// Device/Application/CAN_Rx/CAN0_RX_Inverters
(* VERSION V1_0  *)

FUNCTION_BLOCK CAN0_RX_Inverters
VAR_INPUT
END_VAR
VAR_OUTPUT	
(*INVERTER 1*)
	(* AMK_Actual_Values_1_INV1, ID=283*)
		AMK_bSystemReady1_CAN: BOOL;
		AMK_bError1_CAN: BOOL;
		AMK_bWarn1_CAN: BOOL;
		AMK_bQuitDcOn1_CAN: BOOL;
		AMK_bDcOn1_check_CAN: BOOL;
		AMK_bQuitInverterOn1_CAN: BOOL;
		AMK_bInverterOn1_check_CAN: BOOL;
		AMK_bDerating1_CAN: BOOL;
		AMK_ActualVelocity1_CAN: INT;
		AMK_TorqueCurrent1_CAN: INT;
		AMK_MagnetizingCurrent1_CAN: INT;
	(* AMK_Actual_Values_2_INV1, ID=285*)
		AMK_TempMotor1_CAN: INT;
		AMK_TempInverter1_CAN: INT;
		AMK_ErrorInfo1_CAN: UINT;
		AMK_TempIGBT1_CAN: INT;
(*INVERTER 2*)
	(* AMK_Actual_Values_1_INV2, ID=284*)
		AMK_bSystemReady2_CAN: BOOL;
		AMK_bError2_CAN: BOOL;
		AMK_bWarn2_CAN: BOOL;
		AMK_bQuitDcOn2_CAN: BOOL;
		AMK_bDcOn2_check_CAN: BOOL;
		AMK_bQuitInverterOn2_CAN: BOOL;
		AMK_bInverterOn2_check_CAN: BOOL;
		AMK_bDerating2_CAN: BOOL;
		AMK_ActualVelocity2_CAN: INT;
		AMK_TorqueCurrent2_CAN: INT;
		AMK_MagnetizingCurrent2_CAN: INT;
	(* AMK_Actual_Values_2_INV2, ID=286*)	
		AMK_TempMotor2_CAN: INT;
		AMK_TempInverter2_CAN: INT;
		AMK_ErrorInfo2_CAN: UINT;
		AMK_TempIGBT2_CAN: INT;
(*INVERTER 3*)
	(* AMK_Actual_Values_1_INV3, ID=287*)
		AMK_bSystemReady3_CAN: BOOL;
		AMK_bError3_CAN: BOOL;
		AMK_bWarn3_CAN: BOOL;
		AMK_bQuitDcOn3_CAN: BOOL;
		AMK_bDcOn3_check_CAN: BOOL;
		AMK_bQuitInverterOn3_CAN: BOOL;
		AMK_bInverterOn3_check_CAN: BOOL;
		AMK_bDerating3_CAN: BOOL;
		AMK_ActualVelocity3_CAN: INT;
		AMK_TorqueCurrent3_CAN: INT;
		AMK_MagnetizingCurrent3_CAN: INT;
	(* AMK_Actual_Values_2_INV3, ID=289*)
		AMK_TempMotor3_CAN: INT;
		AMK_TempInverter3_CAN: INT;
		AMK_ErrorInfo3_CAN: UINT;
		AMK_TempIGBT3_CAN: INT;
(*INVERTER 4*)
	(* AMK_Actual_Values_1_INV4, ID=288*)
		AMK_bSystemReady4_CAN: BOOL;
		AMK_bError4_CAN: BOOL;
		AMK_bWarn4_CAN: BOOL;
		AMK_bQuitDcOn4_CAN: BOOL;
		AMK_bDcOn4_check_CAN: BOOL;
		AMK_bQuitInverterOn4_CAN: BOOL;
		AMK_bInverterOn4_check_CAN: BOOL;
		AMK_bDerating4_CAN: BOOL;
		AMK_ActualVelocity4_CAN: INT;
		AMK_TorqueCurrent4_CAN: INT;
		AMK_MagnetizingCurrent4_CAN: INT;
	(* AMK_Actual_Values_2_INV4, ID=290*)
		AMK_TempMotor4_CAN: INT;
		AMK_TempInverter4_CAN: INT;
		AMK_ErrorInfo4_CAN: UINT;
		AMK_TempIGBT4_CAN: INT;
		
		(*
(*DATA_LOGGER*)
		DL_Msg_Cntr_CAN: SINT;
		DL_Status_CAN: SINT;
		DL_Power_CAN: INT;
		DL_Voltage_CAN: INT;
		DL_Current_CAN: INT;
		
(*BATTERY*)
	BatCurrent_MSB_CAN: INT;
	BatVoltage_MSB_CAN: INT;
	BatSoc_CAN: INT;
	BatSoh_CAN: INT;
	BatState_CAN: INT;
	BatAlmLv_CAN: INT;
	BatLife_CAN: INT;
	MaxCellVolt_MSB_CAN: INT;
	MinCellVolt_MSB_CAN: INT;
	MaxCellVoltNO_CAN: INT;
	MinCellVoltNO_CAN: INT;
	MaxTemp_CAN: INT;
	MinTemp_CAN: INT;
	MaxTempNo_CAN: INT;
	MinTempNo_CAN: INT;
	CoolingCtl_CAN: INT;
	HeatingCtl_CAN: INT;
	PosRlyStr_CAN: INT;
	NegRlyStr_CAN: INT;
	PreRlyStr_CAN: INT;
	OnChrRlyStr_CAN: INT;
	OffChrRlyStr_CAN: INT;
	ChrState_CAN: INT;
	ChrCommunication_CAN: BOOL;
	ChrOFFCC2_CAN: BOOL;
	ChrONCC_CAN: INT;
	ChrReqVolt_MSB_CAN: INT;
	ChrReqCurr_MSB_CAN: INT;
	MaxChrCurtLimit_MSB_CAN: INT;
	MaxDisCurtLimit_MSB_CAN: INT;
	MaxChrPowerLimit_MSB_CAN: INT;
	MaxDisPowerLimit_MSB_CAN: INT;
	ALM_CELL_OV_CAN: INT;
	ALM_CELL_UV_CAN: INT;
	ALM_CELL_OT_CAN: INT;
	ALM_CELL_UT_CAN: INT;
	ALM_CELL_LBK_CAN: BOOL;
	ALM_CELL_TBK_CAN: BOOL;
	ALM_BATT_DV_CAN: INT;
	ALM_BATT_DT_CAN: INT;
	ALM_BATT_OV_CAN: INT;
	ALM_BATT_UV_CAN: INT;
	ALM_BATT_OC_CAN: INT;
	ALM_BATT_UC_CAN: INT;
	ALM_CHRG_OCS_CAN: INT;
	ALM_DSCH_OCS_CAN: INT;
	ALM_CHRG_OCT_CAN: INT;
	ALM_DSCH_OCT_CAN: INT;
	ALM_BSU_OFFLINE_CAN: INT;
	ALM_BSU_FAULT_CAN: BOOL;
	ALM_LEAK_OC_CAN: INT;
	ALM_PRECHRG_FAIL_CAN: BOOL;
	ALM_AUX_FAIL_CAN: BOOL;
	ALM_BMU_FAIL_CAN: BOOL;
	ALM_VCU_OFFLINE_CAN: INT;
	ALM_HVREL_FAIL_CAN: BOOL;
	ALM_HALL_BREAK_CAN: BOOL;
	CellVoltN_1_CAN: INT;
	CellVoltN_2_CAN: INT;
	CellVoltN_3_CAN: INT;
	CellVoltN_4_CAN: INT;
	CellVoltN_5_CAN: INT;
	CellVoltN_6_CAN: INT;
	CellVoltN_7_CAN: INT;
	CellVoltN_8_CAN: INT;
	CellVoltN_9_CAN: INT;
	CellVoltN_10_CAN: INT;
	CellVoltN_11_CAN: INT;
	CellVoltN_12_CAN: INT;
	CellVoltN_13_CAN: INT;
	CellVoltN_14_CAN: INT;
	CellVoltN_15_CAN: INT;
	CellVoltN_16_CAN: INT;
	CellVoltN_17_CAN: INT;
	CellVoltN_18_CAN: INT;
	CellVoltN_19_CAN: INT;
	CellVoltN_20_CAN: INT;
	CellVoltN_21_CAN: INT;
	CellVoltN_22_CAN: INT;
	CellVoltN_23_CAN: INT;
	CellVoltN_24_CAN: INT;
	CellVoltN_25_CAN: INT;
	CellVoltN_26_CAN: INT;
	CellVoltN_27_CAN: INT;
	CellVoltN_28_CAN: INT;
	CellVoltN_29_CAN: INT;
	CellVoltN_30_CAN: INT;
	CellVoltN_31_CAN: INT;
	CellVoltN_32_CAN: INT;
	CellVoltN_33_CAN: INT;
	CellVoltN_34_CAN: INT;
	CellVoltN_35_CAN: INT;
	CellVoltN_36_CAN: INT;
	CellVoltN_37_CAN: INT;
	CellVoltN_38_CAN: INT;
	CellVoltN_39_CAN: INT;
	CellVoltN_40_CAN: INT;
	CellVoltN_41_CAN: INT;
	CellVoltN_42_CAN: INT;
	CellVoltN_43_CAN: INT;
	CellVoltN_44_CAN: INT;
	CellVoltN_45_CAN: INT;
	CellVoltN_46_CAN: INT;
	CellVoltN_47_CAN: INT;
	CellVoltN_48_CAN: INT;
	CellVoltN_49_CAN: INT;
	CellVoltN_50_CAN: INT;
	CellVoltN_51_CAN: INT;
	CellVoltN_52_CAN: INT;
	CellVoltN_53_CAN: INT;
	CellVoltN_54_CAN: INT;
	CellVoltN_55_CAN: INT;
	CellVoltN_56_CAN: INT;
	CellVoltN_57_CAN: INT;
	CellVoltN_58_CAN: INT;
	CellVoltN_59_CAN: INT;
	CellVoltN_60_CAN: INT;
	CellVoltN_61_CAN: INT;
	CellVoltN_62_CAN: INT;
	CellVoltN_63_CAN: INT;
	CellVoltN_64_CAN: INT;
	CellVoltN_65_CAN: INT;
	CellVoltN_66_CAN: INT;
	CellVoltN_67_CAN: INT;
	CellVoltN_68_CAN: INT;
	CellVoltN_69_CAN: INT;
	CellVoltN_70_CAN: INT;
	CellVoltN_71_CAN: INT;
	CellVoltN_72_CAN: INT;
	CellVoltN_73_CAN: INT;
	CellVoltN_74_CAN: INT;
	CellVoltN_75_CAN: INT;
	CellVoltN_76_CAN: INT;
	CellVoltN_77_CAN: INT;
	CellVoltN_78_CAN: INT;
	CellVoltN_79_CAN: INT;
	CellVoltN_80_CAN: INT;
	CellVoltN_81_CAN: INT;
	CellVoltN_82_CAN: INT;
	CellVoltN_83_CAN: INT;
	CellVoltN_84_CAN: INT;
	CellVoltN_85_CAN: INT;
	CellVoltN_86_CAN: INT;
	CellVoltN_87_CAN: INT;
	CellVoltN_88_CAN: INT;
	CellVoltN_89_CAN: INT;
	CellVoltN_90_CAN: INT;
	CellVoltN_91_CAN: INT;
	CellVoltN_92_CAN: INT;
	CellVoltN_93_CAN: INT;
	CellVoltN_94_CAN: INT;
	CellVoltN_95_CAN: INT;
	CellVoltN_96_CAN: INT;
	CellVoltN_97_CAN: INT;
	CellVoltN_98_CAN: INT;
	CellVoltN_99_CAN: INT;
	CellVoltN_100_CAN: INT;
	CellVoltN_101_CAN: INT;
	CellVoltN_102_CAN: INT;
	CellVoltN_103_CAN: INT;
	CellVoltN_104_CAN: INT;
	CellVoltN_105_CAN: INT;
	CellVoltN_106_CAN: INT;
	CellVoltN_107_CAN: INT;
	CellVoltN_108_CAN: INT;
	CellVoltN_109_CAN: INT;
	CellVoltN_110_CAN: INT;
	CellVoltN_111_CAN: INT;
	CellVoltN_112_CAN: INT;
	CellVoltN_113_CAN: INT;
	CellVoltN_114_CAN: INT;
	CellVoltN_115_CAN: INT;
	CellVoltN_116_CAN: INT;
	CellVoltN_117_CAN: INT;
	CellVoltN_118_CAN: INT;
	CellVoltN_119_CAN: INT;
	CellVoltN_120_CAN: INT;
	CellVoltN_121_CAN: INT;
	CellVoltN_122_CAN: INT;
	CellVoltN_123_CAN: INT;
	CellVoltN_124_CAN: INT;
	CellVoltN_125_CAN: INT;
	CellVoltN_126_CAN: INT;
	CellVoltN_127_CAN: INT;
	CellVoltN_128_CAN: INT;
	CellVoltN_129_CAN: INT;
	CellVoltN_130_CAN: INT;
	CellVoltN_131_CAN: INT;
	CellVoltN_132_CAN: INT;
	CellVoltN_133_CAN: INT;
	CellVoltN_134_CAN: INT;
	CellVoltN_135_CAN: INT;
	CellVoltN_136_CAN: INT;
	CellVoltN_137_CAN: INT;
	CellVoltN_138_CAN: INT;
	CellTempN_1_CAN: INT;
	CellTempN_2_CAN: INT;
	CellTempN_3_CAN: INT;
	CellTempN_4_CAN: INT;
	CellTempN_5_CAN: INT;
	CellTempN_6_CAN: INT;
	CellTempN_7_CAN: INT;
	CellTempN_8_CAN: INT;
	CellTempN_9_CAN: INT;
	CellTempN_10_CAN: INT;
	CellTempN_11_CAN: INT;
	CellTempN_12_CAN: INT;
	CellTempN_13_CAN: INT;
	CellTempN_14_CAN: INT;
	CellTempN_15_CAN: INT;
	CellTempN_16_CAN: INT;
	CellTempN_17_CAN: INT;
	CellTempN_18_CAN: INT;
	CellTempN_19_CAN: INT;
	CellTempN_20_CAN: INT;
	CellTempN_21_CAN: INT;
	CellTempN_22_CAN: INT;
	CellTempN_23_CAN: INT;
	CellTempN_24_CAN: INT;
	CellTempN_25_CAN: INT;
	CellTempN_26_CAN: INT;
	CellTempN_27_CAN: INT;
	CellTempN_28_CAN: INT;
	CellTempN_29_CAN: INT;
	CellTempN_30_CAN: INT;
	CellTempN_31_CAN: INT;
	CellTempN_32_CAN: INT;
	CellTempN_33_CAN: INT;
	CellTempN_34_CAN: INT;
	CellTempN_35_CAN: INT;
	CellTempN_36_CAN: INT;
	CellTempN_37_CAN: INT;
	CellTempN_38_CAN: INT;
	CellTempN_39_CAN: INT;
	CellTempN_40_CAN: INT;
	CellTempN_41_CAN: INT;
	CellTempN_42_CAN: INT;
	CellTempN_43_CAN: INT;
	CellTempN_44_CAN: INT;
	CellTempN_45_CAN: INT;
	CellTempN_46_CAN: INT;
	CellTempN_47_CAN: INT;
	CellTempN_48_CAN: INT;
	CellTempN_49_CAN: INT;
	CellTempN_50_CAN: INT;
	CellTempN_51_CAN: INT;
	CellTempN_52_CAN: INT;
	CellTempN_53_CAN: INT;
	CellTempN_54_CAN: INT;
	CellTempN_55_CAN: INT;
	CellTempN_56_CAN: INT;
	CellTempN_57_CAN: INT;
	CellTempN_58_CAN: INT;
	CellTempN_59_CAN: INT;
	CellTempN_60_CAN: INT;
	MainRlyCmd_CAN: INT;
	ShutDownCmd_CAN: INT;
	BMS_State_CAN: DINT;
	*)
			
END_VAR
VAR
(*CanRx*)
	(* INVERTER_1*)
		FBRX_AMK_Actual_Values_1_INV1: CanRx;
		FBRX_AMK_Actual_Values_2_INV1: CanRx;
	(* INVERTER_2*)
		FBRX_AMK_Actual_Values_1_INV2:CanRx;
		FBRX_AMK_Actual_Values_2_INV2:CanRx;
	(* INVERTER_3*)
		FBRX_AMK_Actual_Values_1_INV3:CanRx;
		FBRX_AMK_Actual_Values_2_INV3:CanRx;
	(* INVERTER_4*)
		FBRX_AMK_Actual_Values_1_INV4:CanRx;
		FBRX_AMK_Actual_Values_2_INV4:CanRx;
		
		(*
	(*BATTERY*)
		FBRX_BATTERY:CanRx;
	(*DATA_LOGGER*)	
		FBRX_DATA_LOGGER:CanRx;
		
		(*BATTERY*)
		FBRX_BMS_HCU_INFO:CanRx;
		FBRX_BMS_HCU_MAXV: CanRx;
		FBRX_BMS_HCU_MAXT: CanRx;
		FBRX_BMS_HCU_RELAY: CanRx;
		FBRX_BMS_HCU_POWER: CanRx;
		FBRX_BMS_HCU_ALARM: CanRx;
		FBRX_BMS_HCU_CMD: CanRx;
		FBRX_BMS_HCU_CELLV_1: CanRx;
		FBRX_BMS_HCU_CELLV_2: CanRx;
		FBRX_BMS_HCU_CELLV_3: CanRx;
		FBRX_BMS_HCU_CELLV_4: CanRx;
		FBRX_BMS_HCU_CELLV_5: CanRx;
		FBRX_BMS_HCU_CELLV_6: CanRx;
		FBRX_BMS_HCU_CELLV_7: CanRx;
		FBRX_BMS_HCU_CELLV_8: CanRx;
		FBRX_BMS_HCU_CELLV_9: CanRx;
		FBRX_BMS_HCU_CELLV_10: CanRx;
		FBRX_BMS_HCU_CELLV_11: CanRx;
		FBRX_BMS_HCU_CELLV_12: CanRx;
		FBRX_BMS_HCU_CELLV_13: CanRx;
		FBRX_BMS_HCU_CELLV_14: CanRx;
		FBRX_BMS_HCU_CELLV_15: CanRx;
		FBRX_BMS_HCU_CELLV_16: CanRx;
		FBRX_BMS_HCU_CELLV_17: CanRx;
		FBRX_BMS_HCU_CELLV_18: CanRx;
		FBRX_BMS_HCU_CELLV_19: CanRx;
		FBRX_BMS_HCU_CELLV_20: CanRx;
		FBRX_BMS_HCU_CELLV_21: CanRx;
		FBRX_BMS_HCU_CELLV_22: CanRx;
		FBRX_BMS_HCU_CELLV_23: CanRx;
		FBRX_BMS_HCU_CELLV_24: CanRx;
		FBRX_BMS_HCU_CELLV_25: CanRx;
		FBRX_BMS_HCU_CELLV_26: CanRx;
		FBRX_BMS_HCU_CELLV_27: CanRx;
		FBRX_BMS_HCU_CELLV_28: CanRx;
		FBRX_BMS_HCU_CELLV_29: CanRx;
		FBRX_BMS_HCU_CELLV_30: CanRx;
		FBRX_BMS_HCU_CELLV_31: CanRx;
		FBRX_BMS_HCU_CELLV_32: CanRx;
		FBRX_BMS_HCU_CELLV_33: CanRx;
		FBRX_BMS_HCU_CELLV_34: CanRx;
		FBRX_BMS_HCU_CELLV_35: CanRx;
		FBRX_BMS_HCU_CELLT_1: CanRx;
		FBRX_BMS_HCU_CELLT_2: CanRx;
		FBRX_BMS_HCU_CELLT_3: CanRx;
		FBRX_BMS_HCU_CELLT_4: CanRx;
		FBRX_BMS_HCU_CELLT_5: CanRx;
		FBRX_BMS_HCU_CELLT_6: CanRx;
		FBRX_BMS_HCU_CELLT_7: CanRx;
		FBRX_BMS_HCU_CELLT_8: CanRx;
		FBRX_Battery_status: CanRx;
		*)
		
(*Time_out_Counter*)
	(* INVERTER_1*)
		Counter_time_out_AMK_Actual_Values_1_INV1:INT:=0;
		Counter_time_out_AMK_Actual_Values_2_INV1:INT:=0;
	(* INVERTER_2*)	
		Counter_time_out_AMK_Actual_Values_1_INV2:INT:=0;
		Counter_time_out_AMK_Actual_Values_2_INV2:INT:=0;
	(* INVERTER_3*)	
		Counter_time_out_AMK_Actual_Values_1_INV3:INT:=0;
		Counter_time_out_AMK_Actual_Values_2_INV3:INT:=0;
	(* INVERTER_4*)	
		Counter_time_out_AMK_Actual_Values_1_INV4:INT:=0;
		Counter_time_out_AMK_Actual_Values_2_INV4:INT:=0;
		(*
	(*battery*)
		Counter_time_out_BATTERY:INT:=0;
		Counter_time_out_FBRX_BMS_HCU_INFO:INT:=0;
	(*DATA_LOGGER*)
		Counter_time_out_DATA_LOGGER:INT:=0;	
		
		*)
		
		
END_VAR

(*--------------------------------------------------INVERTER_1_RX--------------------------------------------------*)
	(* AMK_Actual_Values_1_INV1, ID=283*)
		FBRX_AMK_Actual_Values_1_INV1 (	iCAN			:= ADR(GVL.H_CAN_RX_0),  				(* Structure for sending / receiving CAN messages *)
								iCanId				:= 16#283,							(* CAN Id of receiving message *) 
								iCanIdExtended		:= FALSE,  							(* Standard CAN Frame *)
								iTimeoutLimit		:= T#500MS,							(* Timeout after 500ms - Flag will be set *) 
								oByteCount			=> , 
								oData				=> , 
								oNewData			=> , 
								oCanTimeout			=> , 
								oReceiverId			=> , 
								oTooManyReceivers	=> );	
				
								
				IF FBRX_AMK_Actual_Values_1_INV1  .oNewData THEN											(* If new CAN data is available *)
						AMK_bSystemReady1_CAN:=FBRX_AMK_Actual_Values_1_INV1.oData[1].0;
						AMK_bError1_CAN:=FBRX_AMK_Actual_Values_1_INV1.oData[1].1;
						AMK_bWarn1_CAN:=FBRX_AMK_Actual_Values_1_INV1.oData[1].2;
						AMK_bQuitDcOn1_CAN:=FBRX_AMK_Actual_Values_1_INV1.oData[1].3;
						AMK_bDcOn1_check_CAN:=FBRX_AMK_Actual_Values_1_INV1.oData[1].4;
						AMK_bQuitInverterOn1_CAN:=FBRX_AMK_Actual_Values_1_INV1.oData[1].5;
						AMK_bInverterOn1_check_CAN:=FBRX_AMK_Actual_Values_1_INV1.oData[1].6;
						AMK_bDerating1_CAN:=FBRX_AMK_Actual_Values_1_INV1.oData[1].7;
						AMK_ActualVelocity1_CAN:=FBRX_AMK_Actual_Values_1_INV1.oData[2]+SHL(BYTE_TO_INT(FBRX_AMK_Actual_Values_1_INV1.oData[3]),8);
						AMK_TorqueCurrent1_CAN:=FBRX_AMK_Actual_Values_1_INV1.oData[4]+SHL(BYTE_TO_INT(FBRX_AMK_Actual_Values_1_INV1.oData[5]),8);
						AMK_MagnetizingCurrent1_CAN:=FBRX_AMK_Actual_Values_1_INV1.oData[6]+SHL(BYTE_TO_INT(FBRX_AMK_Actual_Values_1_INV1.oData[7]),8);
				ELSIF FBRX_AMK_Actual_Values_1_INV1 .oCanTimeout THEN										(* If timeout flag is enabled switch off LedRed *)
				 (*Crear los errores necesarios para cuando no se leen las variable despues del time out*)
						Counter_time_out_AMK_Actual_Values_1_INV1:=Counter_time_out_AMK_Actual_Values_1_INV1+1;
				END_IF 
	(* AMK_Actual_Values_2_INV1, ID=285*)
			FBRX_AMK_Actual_Values_2_INV1 (	iCAN			:= ADR(GVL.H_CAN_RX_0),  				(* Structure for sending / receiving CAN messages *)
								iCanId				:= 16#285,							(* CAN Id of receiving message *) 
								iCanIdExtended		:= FALSE,  							(* Standard CAN Frame *)
								iTimeoutLimit		:= T#500MS,							(* Timeout after 500ms - Flag will be set *) 
								oByteCount			=> , 
								oData				=> , 
								oNewData			=> , 
								oCanTimeout			=> , 
								oReceiverId			=> , 
								oTooManyReceivers	=> );	
				
								
				IF FBRX_AMK_Actual_Values_2_INV1  .oNewData THEN											(* If new CAN data is available *)
						AMK_TempMotor1_CAN:=FBRX_AMK_Actual_Values_2_INV1.oData[0]+SHL(BYTE_TO_INT(FBRX_AMK_Actual_Values_2_INV1.oData[1]),8);
						AMK_TempInverter1_CAN:=FBRX_AMK_Actual_Values_2_INV1.oData[2]+SHL(BYTE_TO_INT(FBRX_AMK_Actual_Values_2_INV1.oData[3]),8);
						AMK_ErrorInfo1_CAN:=FBRX_AMK_Actual_Values_2_INV1.oData[4]+SHL(BYTE_TO_UINT(FBRX_AMK_Actual_Values_2_INV1.oData[5]),8);
						
						AMK_TempIGBT1_CAN:=FBRX_AMK_Actual_Values_2_INV1.oData[6]+SHL(BYTE_TO_INT(FBRX_AMK_Actual_Values_2_INV1.oData[7]),8);
				ELSIF FBRX_AMK_Actual_Values_2_INV1 .oCanTimeout THEN										(* If timeout flag is enabled switch off LedRed *)
				 (*Crear los errores necesarios para cuando no se leen las variable despues del time out*)
						Counter_time_out_AMK_Actual_Values_2_INV1:=Counter_time_out_AMK_Actual_Values_2_INV1+1;
				END_IF
(*-----------------------------------------------FIN_INVERTER_1_RX--------------------------------------------------*)


(*--------------------------------------------------INVERTER_2_RX--------------------------------------------------*)
	(* AMK_Actual_Values_1_INV2, ID=284*)
		FBRX_AMK_Actual_Values_1_INV2 (	iCAN			:= ADR(GVL.H_CAN_RX_0),  				(* Structure for sending / receiving CAN messages *)
								iCanId				:= 16#284,							(* CAN Id of receiving message *) 
								iCanIdExtended		:= FALSE,  							(* Standard CAN Frame *)
								iTimeoutLimit		:= T#500MS,							(* Timeout after 500ms - Flag will be set *) 
								oByteCount			=> , 
								oData				=> , 
								oNewData			=> , 
								oCanTimeout			=> , 
								oReceiverId			=> , 
								oTooManyReceivers	=> );	
				
								
				IF FBRX_AMK_Actual_Values_1_INV2  .oNewData THEN											(* If new CAN data is available *)
						AMK_bSystemReady2_CAN:=FBRX_AMK_Actual_Values_1_INV2.oData[1].0;
						AMK_bError2_CAN:=FBRX_AMK_Actual_Values_1_INV2.oData[1].1;
						AMK_bWarn2_CAN:=FBRX_AMK_Actual_Values_1_INV2.oData[1].2;
						AMK_bQuitDcOn2_CAN:=FBRX_AMK_Actual_Values_1_INV2.oData[1].3;
						AMK_bDcOn2_check_CAN:=FBRX_AMK_Actual_Values_1_INV2.oData[1].4;
						AMK_bQuitInverterOn2_CAN:=FBRX_AMK_Actual_Values_1_INV2.oData[1].5;
						AMK_bInverterOn2_check_CAN:=FBRX_AMK_Actual_Values_1_INV2.oData[1].6;
						AMK_bDerating2_CAN:=FBRX_AMK_Actual_Values_1_INV2.oData[1].7;
						AMK_ActualVelocity2_CAN:=FBRX_AMK_Actual_Values_1_INV2.oData[2]+SHL(BYTE_TO_INT(FBRX_AMK_Actual_Values_1_INV2.oData[3]),8);
						AMK_TorqueCurrent2_CAN:=FBRX_AMK_Actual_Values_1_INV2.oData[4]+SHL(BYTE_TO_INT(FBRX_AMK_Actual_Values_1_INV2.oData[5]),8);
						AMK_MagnetizingCurrent2_CAN:=FBRX_AMK_Actual_Values_1_INV2.oData[6]+SHL(BYTE_TO_INT(FBRX_AMK_Actual_Values_1_INV2.oData[7]),8);
				ELSIF FBRX_AMK_Actual_Values_1_INV2 .oCanTimeout THEN										(* If timeout flag is enabled switch off LedRed *)
				 (*Crear los errores necesarios para cuando no se leen las variable despues del time out*)
						Counter_time_out_AMK_Actual_Values_1_INV2:=Counter_time_out_AMK_Actual_Values_1_INV2+1;
				END_IF
	(* AMK_Actual_Values_2_INV2, ID=286*)
			FBRX_AMK_Actual_Values_2_INV2 (	iCAN			:= ADR(GVL.H_CAN_RX_0),  				(* Structure for sending / receiving CAN messages *)
								iCanId				:= 16#286,							(* CAN Id of receiving message *) 
								iCanIdExtended		:= FALSE,  							(* Standard CAN Frame *)
								iTimeoutLimit		:= T#500MS,							(* Timeout after 500ms - Flag will be set *) 
								oByteCount			=> , 
								oData				=> , 
								oNewData			=> , 
								oCanTimeout			=> , 
								oReceiverId			=> , 
								oTooManyReceivers	=> );	
				
								
				IF FBRX_AMK_Actual_Values_2_INV2  .oNewData THEN											(* If new CAN data is available *)
						AMK_TempMotor2_CAN:=FBRX_AMK_Actual_Values_2_INV2.oData[0]+SHL(BYTE_TO_INT(FBRX_AMK_Actual_Values_2_INV2.oData[1]),8);
						AMK_TempInverter2_CAN:=FBRX_AMK_Actual_Values_2_INV2.oData[2]+SHL(BYTE_TO_INT(FBRX_AMK_Actual_Values_2_INV2.oData[3]),8);
						AMK_ErrorInfo2_CAN:=FBRX_AMK_Actual_Values_2_INV2.oData[4]+SHL(BYTE_TO_UINT(FBRX_AMK_Actual_Values_2_INV2.oData[5]),8);
						AMK_TempIGBT2_CAN:=FBRX_AMK_Actual_Values_2_INV2.oData[6]+SHL(BYTE_TO_INT(FBRX_AMK_Actual_Values_2_INV2.oData[7]),8);
				ELSIF FBRX_AMK_Actual_Values_2_INV2 .oCanTimeout THEN										(* If timeout flag is enabled switch off LedRed *)
				 (*Crear los errores necesarios para cuando no se leen las variable despues del time out*)
						Counter_time_out_AMK_Actual_Values_2_INV2:=Counter_time_out_AMK_Actual_Values_2_INV2+1;
				END_IF
(*-----------------------------------------------FIN_INVERTER_2_RX--------------------------------------------------*)


(*--------------------------------------------------INVERTER_3_RX--------------------------------------------------*)
(* AMK_Actual_Values_1_INV3, ID=287*)
		FBRX_AMK_Actual_Values_1_INV3 (	iCAN			:= ADR(GVL.H_CAN_RX_0),  				(* Structure for sending / receiving CAN messages *)
								iCanId				:= 16#287,							(* CAN Id of receiving message *) 
								iCanIdExtended		:= FALSE,  							(* Standard CAN Frame *)
								iTimeoutLimit		:= T#500MS,							(* Timeout after 500ms - Flag will be set *) 
								oByteCount			=> , 
								oData				=> , 
								oNewData			=> , 
								oCanTimeout			=> , 
								oReceiverId			=> , 
								oTooManyReceivers	=> );	
				
								
				IF FBRX_AMK_Actual_Values_1_INV3  .oNewData THEN											(* If new CAN data is available *)
						AMK_bSystemReady3_CAN:=FBRX_AMK_Actual_Values_1_INV3.oData[1].0;
						AMK_bError3_CAN:=FBRX_AMK_Actual_Values_1_INV3.oData[1].1;
						AMK_bWarn3_CAN:=FBRX_AMK_Actual_Values_1_INV3.oData[1].2;
						AMK_bQuitDcOn3_CAN:=FBRX_AMK_Actual_Values_1_INV3.oData[1].3;
						AMK_bDcOn3_check_CAN:=FBRX_AMK_Actual_Values_1_INV3.oData[1].4;
						AMK_bQuitInverterOn3_CAN:=FBRX_AMK_Actual_Values_1_INV3.oData[1].5;
						AMK_bInverterOn3_check_CAN:=FBRX_AMK_Actual_Values_1_INV3.oData[1].6;
						AMK_bDerating3_CAN:=FBRX_AMK_Actual_Values_1_INV3.oData[1].7;
						AMK_ActualVelocity3_CAN:=FBRX_AMK_Actual_Values_1_INV3.oData[2]+SHL(BYTE_TO_INT(FBRX_AMK_Actual_Values_1_INV3.oData[3]),8);
						AMK_TorqueCurrent3_CAN:=FBRX_AMK_Actual_Values_1_INV3.oData[4]+SHL(BYTE_TO_INT(FBRX_AMK_Actual_Values_1_INV3.oData[5]),8);
						AMK_MagnetizingCurrent3_CAN:=FBRX_AMK_Actual_Values_1_INV3.oData[6]+SHL(BYTE_TO_INT(FBRX_AMK_Actual_Values_1_INV3.oData[7]),8);
				ELSIF FBRX_AMK_Actual_Values_1_INV3 .oCanTimeout THEN										(* If timeout flag is enabled switch off LedRed *)
				 (*Crear los errores necesarios para cuando no se leen las variable despues del time out*)
						Counter_time_out_AMK_Actual_Values_1_INV3:=Counter_time_out_AMK_Actual_Values_1_INV3+1;
				END_IF
(* AMK_Actual_Values_2_INV3, ID=289*)
			FBRX_AMK_Actual_Values_2_INV3 (	iCAN			:= ADR(GVL.H_CAN_RX_0),  				(* Structure for sending / receiving CAN messages *)
								iCanId				:= 16#289,							(* CAN Id of receiving message *) 
								iCanIdExtended		:= FALSE,  							(* Standard CAN Frame *)
								iTimeoutLimit		:= T#500MS,							(* Timeout after 500ms - Flag will be set *) 
								oByteCount			=> , 
								oData				=> , 
								oNewData			=> , 
								oCanTimeout			=> , 
								oReceiverId			=> , 
								oTooManyReceivers	=> );	
				
								
				IF FBRX_AMK_Actual_Values_2_INV3  .oNewData THEN											(* If new CAN data is available *)
						AMK_TempMotor3_CAN:=FBRX_AMK_Actual_Values_2_INV3.oData[0]+SHL(BYTE_TO_INT(FBRX_AMK_Actual_Values_2_INV3.oData[1]),8);
						AMK_TempInverter3_CAN:=FBRX_AMK_Actual_Values_2_INV3.oData[2]+SHL(BYTE_TO_INT(FBRX_AMK_Actual_Values_2_INV3.oData[3]),8);
						AMK_ErrorInfo3_CAN:=FBRX_AMK_Actual_Values_2_INV3.oData[4]+SHL(BYTE_TO_UINT(FBRX_AMK_Actual_Values_2_INV3.oData[5]),8);
						AMK_TempIGBT3_CAN:=FBRX_AMK_Actual_Values_2_INV3.oData[6]+SHL(BYTE_TO_INT(FBRX_AMK_Actual_Values_2_INV3.oData[7]),8);
				ELSIF FBRX_AMK_Actual_Values_2_INV3 .oCanTimeout THEN										(* If timeout flag is enabled switch off LedRed *)
				 (*Crear los errores necesarios para cuando no se leen las variable despues del time out*)
						Counter_time_out_AMK_Actual_Values_2_INV3:=Counter_time_out_AMK_Actual_Values_2_INV3+1;
				END_IF
(*-----------------------------------------------FIN_INVERTER_3_RX--------------------------------------------------*)



(*--------------------------------------------------INVERTER_4_RX--------------------------------------------------*)
	(* AMK_Actual_Values_1_INV4, ID=288*)
		FBRX_AMK_Actual_Values_1_INV4 (	iCAN			:= ADR(GVL.H_CAN_RX_0),  				(* Structure for sending / receiving CAN messages *)
								iCanId				:= 16#288,							(* CAN Id of receiving message *) 
								iCanIdExtended		:= FALSE,  							(* Standard CAN Frame *)
								iTimeoutLimit		:= T#500MS,							(* Timeout after 500ms - Flag will be set *) 
								oByteCount			=> , 
								oData				=> , 
								oNewData			=> , 
								oCanTimeout			=> , 
								oReceiverId			=> , 
								oTooManyReceivers	=> );	
				
								
				IF FBRX_AMK_Actual_Values_1_INV4  .oNewData THEN											(* If new CAN data is available *)
						AMK_bSystemReady4_CAN:=FBRX_AMK_Actual_Values_1_INV4.oData[1].0;
						AMK_bError4_CAN:=FBRX_AMK_Actual_Values_1_INV4.oData[1].1;
						AMK_bWarn4_CAN:=FBRX_AMK_Actual_Values_1_INV4.oData[1].2;
						AMK_bQuitDcOn4_CAN:=FBRX_AMK_Actual_Values_1_INV4.oData[1].3;
						AMK_bDcOn4_check_CAN:=FBRX_AMK_Actual_Values_1_INV4.oData[1].4;
						AMK_bQuitInverterOn4_CAN:=FBRX_AMK_Actual_Values_1_INV4.oData[1].5;
						AMK_bInverterOn4_check_CAN:=FBRX_AMK_Actual_Values_1_INV4.oData[1].6;
						AMK_bDerating4_CAN:=FBRX_AMK_Actual_Values_1_INV4.oData[1].7;
						AMK_ActualVelocity4_CAN:=FBRX_AMK_Actual_Values_1_INV4.oData[2]+SHL(BYTE_TO_INT(FBRX_AMK_Actual_Values_1_INV4.oData[3]),8);
						AMK_TorqueCurrent4_CAN:=FBRX_AMK_Actual_Values_1_INV4.oData[4]+SHL(BYTE_TO_INT(FBRX_AMK_Actual_Values_1_INV4.oData[5]),8);
						AMK_MagnetizingCurrent4_CAN:=FBRX_AMK_Actual_Values_1_INV4.oData[6]+SHL(BYTE_TO_INT(FBRX_AMK_Actual_Values_1_INV4.oData[7]),8);
				ELSIF FBRX_AMK_Actual_Values_1_INV4 .oCanTimeout THEN										(* If timeout flag is enabled switch off LedRed *)
				 (*Crear los errores necesarios para cuando no se leen las variable despues del time out*)
						Counter_time_out_AMK_Actual_Values_1_INV4:=Counter_time_out_AMK_Actual_Values_1_INV4+1;
				END_IF
	(* AMK_Actual_Values_2_INV4, ID=290*)
			FBRX_AMK_Actual_Values_2_INV4 (	iCAN			:= ADR(GVL.H_CAN_RX_0),  				(* Structure for sending / receiving CAN messages *)
								iCanId				:= 16#28A,							(* CAN Id of receiving message *) 
								iCanIdExtended		:= FALSE,  							(* Standard CAN Frame *)
								iTimeoutLimit		:= T#500MS,							(* Timeout after 500ms - Flag will be set *) 
								oByteCount			=> , 
								oData				=> , 
								oNewData			=> , 
								oCanTimeout			=> , 
								oReceiverId			=> , 
								oTooManyReceivers	=> );	
				
								
				IF FBRX_AMK_Actual_Values_2_INV4  .oNewData THEN											(* If new CAN data is available *)
						AMK_TempMotor4_CAN:=FBRX_AMK_Actual_Values_2_INV4.oData[0]+SHL(BYTE_TO_INT(FBRX_AMK_Actual_Values_2_INV4.oData[1]),8);
						AMK_TempInverter4_CAN:=FBRX_AMK_Actual_Values_2_INV4.oData[2]+SHL(BYTE_TO_INT(FBRX_AMK_Actual_Values_2_INV4.oData[3]),8);
						AMK_ErrorInfo4_CAN:=FBRX_AMK_Actual_Values_2_INV4.oData[4]+SHL(BYTE_TO_UINT(FBRX_AMK_Actual_Values_2_INV4.oData[5]),8);
						AMK_TempIGBT4_CAN:=FBRX_AMK_Actual_Values_2_INV4.oData[6]+SHL(BYTE_TO_INT(FBRX_AMK_Actual_Values_2_INV4.oData[7]),8);
				ELSIF FBRX_AMK_Actual_Values_2_INV4 .oCanTimeout THEN										(* If timeout flag is enabled switch off LedRed *)
				 (*Crear los errores necesarios para cuando no se leen las variable despues del time out*)
						Counter_time_out_AMK_Actual_Values_2_INV4:=Counter_time_out_AMK_Actual_Values_2_INV4+1;
				END_IF
(*-----------------------------------------------FIN_INVERTER_4_RX--------------------------------------------------*)

(*
(*--------------------------------------------------DATA_LOGGER--------------------------------------------------*)
	(* AMK_Actual_Values_1_INV4, ID=288*)
		FBRX_DATA_LOGGER (	iCAN			:= ADR(GVL.H_CAN_RX_2),  				(* Structure for sending / receiving CAN messages *)
								iCanId				:= 16#430,							(* CAN Id of receiving message *) 
								iCanIdExtended		:= FALSE,  							(* Standard CAN Frame *)
								iTimeoutLimit		:= T#500MS,							(* Timeout after 500ms - Flag will be set *) 
								oByteCount			=> , 
								oData				=> , 
								oNewData			=> , 
								oCanTimeout			=> , 
								oReceiverId			=> , 
								oTooManyReceivers	=> );	
				
								
				IF FBRX_DATA_LOGGER  .oNewData THEN											(* If new CAN data is available *)
						DL_Msg_Cntr_CAN := BYTE_TO_SINT(FBRX_DATA_LOGGER.oData[0]); 
						DL_Status_CAN := BYTE_TO_SINT(FBRX_DATA_LOGGER.oData[1]);  
						DL_Power_CAN := FBRX_DATA_LOGGER.oData[3]+SHL(BYTE_TO_INT(FBRX_DATA_LOGGER.oData[2]),8);
						DL_Voltage_CAN := FBRX_DATA_LOGGER.oData[5]+SHL(BYTE_TO_INT(FBRX_DATA_LOGGER.oData[4]),8);
						DL_Current_CAN := FBRX_DATA_LOGGER.oData[7]+SHL(BYTE_TO_INT(FBRX_DATA_LOGGER.oData[6]),8);
						
						
						
				ELSIF FBRX_DATA_LOGGER .oCanTimeout THEN										(* If timeout flag is enabled switch off LedRed *)
				 (*Crear los errores necesarios para cuando no se leen las variable despues del time out*)
						Counter_time_out_DATA_LOGGER:=Counter_time_out_DATA_LOGGER+1;
				END_IF

(*-----------------------------------------------DATA_LOGGER--------------------------------------------------*)




(*--------------------------------------------------BATTERY_RX--------------------------------------------------*)
	(* BATTERY, ID=170*)
	    FBRX_BMS_HCU_INFO  (	iCAN			:= ADR(GVL.H_CAN_RX_6),  				(* Structure for sending / receiving CAN messages *)
								iCanId				:= 16#186040F3,							(* CAN Id of receiving message *) 
								iCanIdExtended		:= TRUE,  							(* Standard CAN Frame *)
								iTimeoutLimit		:= T#500MS,							(* Timeout after 500ms - Flag will be set *) 
								oByteCount			=> , 
								oData				=> , 
								oNewData			=> , 
								oCanTimeout			=> , 
								oReceiverId			=> , 
								oTooManyReceivers	=> );	
				
								
				IF FBRX_BMS_HCU_INFO   .oNewData THEN											(* If new CAN data is available *)
						
						BatCurrent_MSB_CAN:=FBRX_BMS_HCU_INFO.oData[3]+SHL(BYTE_TO_INT(FBRX_BMS_HCU_INFO.oData[2]),8);
						
						BatVoltage_MSB_CAN:=FBRX_BMS_HCU_INFO.oData[1]+SHL(BYTE_TO_INT(FBRX_BMS_HCU_INFO.oData[0]),8);
						
						BatSoc_CAN:=FBRX_BMS_HCU_INFO.oData[4];
						
						BatSoh_CAN:=FBRX_BMS_HCU_INFO.oData[5];
						
						BatState_CAN:= (BIT_TO_BYTE(FBRX_BMS_HCU_INFO.oData[6].4)+SHL(BIT_TO_BYTE(FBRX_BMS_HCU_INFO.oData[6].5),1)+SHL(BIT_TO_BYTE(FBRX_BMS_HCU_INFO.oData[6].6),2)+SHL(BIT_TO_BYTE(FBRX_BMS_HCU_INFO.oData[6].7),3));
						
						BatAlmLv_CAN:= (BIT_TO_BYTE(FBRX_BMS_HCU_INFO.oData[6].0)+SHL(BIT_TO_BYTE(FBRX_BMS_HCU_INFO.oData[6].1),1)+SHL(BIT_TO_BYTE(FBRX_BMS_HCU_INFO.oData[6].2),2)+SHL(BIT_TO_BYTE(FBRX_BMS_HCU_INFO.oData[6].3),3));  (*Ver como poner la mitad de un byte*)
												
						BatLife_CAN:=FBRX_BMS_HCU_INFO.oData[7];
						
				ELSIF FBRX_BMS_HCU_INFO .oCanTimeout THEN										(* If timeout flag is enabled switch off LedRed *)
				 (*Crear los errores necesarios para cuando no se leen las variable despues del time out*)
						Counter_time_out_FBRX_BMS_HCU_INFO:=Counter_time_out_FBRX_BMS_HCU_INFO+1;
				END_IF
				
		FBRX_BMS_HCU_MAXV  (	iCAN			:= ADR(GVL.H_CAN_RX_6),  				(* Structure for sending / receiving CAN messages *)
								iCanId				:= 16#186140F3,							(* CAN Id of receiving message *) 
								iCanIdExtended		:= TRUE,  							(* Standard CAN Frame *)
								iTimeoutLimit		:= T#500MS,							(* Timeout after 500ms - Flag will be set *) 
								oByteCount			=> , 
								oData				=> , 
								oNewData			=> , 
								oCanTimeout			=> , 
								oReceiverId			=> , 
								oTooManyReceivers	=> );	
				
								
				IF FBRX_BMS_HCU_MAXV   .oNewData THEN											(* If new CAN data is available *)
						
						MaxCellVolt_MSB_CAN:=FBRX_BMS_HCU_MAXV.oData[1]+SHL(BYTE_TO_INT(FBRX_BMS_HCU_MAXV.oData[0]),8);
						MinCellVolt_MSB_CAN:=FBRX_BMS_HCU_MAXV.oData[3]+SHL(BYTE_TO_INT(FBRX_BMS_HCU_MAXV.oData[2]),8);
						MaxCellVoltNO_CAN:=FBRX_BMS_HCU_MAXV.oData[4];
						MinCellVoltNO_CAN:=FBRX_BMS_HCU_MAXV.oData[5];
						
				ELSIF FBRX_BMS_HCU_MAXV .oCanTimeout THEN										(* If timeout flag is enabled switch off LedRed *)
				 (*Crear los errores necesarios para cuando no se leen las variable despues del time out*)
						Counter_time_out_BATTERY:=Counter_time_out_BATTERY+1;
				END_IF
				
	    FBRX_BMS_HCU_MAXT  (	iCAN			:= ADR(GVL.H_CAN_RX_6),  				(* Structure for sending / receiving CAN messages *)
								iCanId				:= 16#186240F3,							(* CAN Id of receiving message *) 
								iCanIdExtended		:= TRUE,  							(* Standard CAN Frame *)
								iTimeoutLimit		:= T#500MS,							(* Timeout after 500ms - Flag will be set *) 
								oByteCount			=> , 
								oData				=> , 
								oNewData			=> , 
								oCanTimeout			=> , 
								oReceiverId			=> , 
								oTooManyReceivers	=> );	
				
								
				IF FBRX_BMS_HCU_MAXT   .oNewData THEN											(* If new CAN data is available *)
						
						MaxTemp_CAN:=FBRX_BMS_HCU_MAXT.oData[0];
						MinTemp_CAN:=FBRX_BMS_HCU_MAXT.oData[1];
						MaxTempNo_CAN:=FBRX_BMS_HCU_MAXT.oData[2];
						MinTempNo_CAN:=FBRX_BMS_HCU_MAXT.oData[3];
						CoolingCtl_CAN:=FBRX_BMS_HCU_MAXT.oData[4];
						HeatingCtl_CAN:=FBRX_BMS_HCU_MAXT.oData[5];
				ELSIF FBRX_BMS_HCU_MAXT .oCanTimeout THEN										(* If timeout flag is enabled switch off LedRed *)
				 (*Crear los errores necesarios para cuando no se leen las variable despues del time out*)
						Counter_time_out_BATTERY:=Counter_time_out_BATTERY+1;
				END_IF
		FBRX_BMS_HCU_RELAY  (	iCAN			:= ADR(GVL.H_CAN_RX_6),  				(* Structure for sending / receiving CAN messages *)
								iCanId				:= 16#186340F3,							(* CAN Id of receiving message *) 
								iCanIdExtended		:= TRUE,  							(* Standard CAN Frame *)
								iTimeoutLimit		:= T#500MS,							(* Timeout after 500ms - Flag will be set *) 
								oByteCount			=> , 
								oData				=> , 
								oNewData			=> , 
								oCanTimeout			=> , 
								oReceiverId			=> , 
								oTooManyReceivers	=> );	
				
								
				IF FBRX_BMS_HCU_RELAY   .oNewData THEN											(* If new CAN data is available *)
						
						PosRlyStr_CAN:= (BIT_TO_BYTE(FBRX_BMS_HCU_RELAY.oData[0].7)+SHL(BIT_TO_BYTE(FBRX_BMS_HCU_RELAY.oData[0].6),1));
						NegRlyStr_CAN:= (BIT_TO_BYTE(FBRX_BMS_HCU_RELAY.oData[0].5)+SHL(BIT_TO_BYTE(FBRX_BMS_HCU_RELAY.oData[0].4),1));
						PreRlyStr_CAN:= (BIT_TO_BYTE(FBRX_BMS_HCU_RELAY.oData[0].3)+SHL(BIT_TO_BYTE(FBRX_BMS_HCU_RELAY.oData[0].2),1));
						OnChrRlyStr_CAN:=(BIT_TO_BYTE(FBRX_BMS_HCU_RELAY.oData[0].1)+SHL(BIT_TO_BYTE(FBRX_BMS_HCU_RELAY.oData[0].0),1));  
						OffChrRlyStr_CAN:= BYTE_TO_SINT(FBRX_BMS_HCU_RELAY.oData[1]);
						ChrState_CAN:= (BIT_TO_BYTE(FBRX_BMS_HCU_RELAY.oData[2].4)+SHL(BIT_TO_BYTE(FBRX_BMS_HCU_RELAY.oData[2].5),1)+SHL(BIT_TO_BYTE(FBRX_BMS_HCU_RELAY.oData[2].6),2)+SHL(BIT_TO_BYTE(FBRX_BMS_HCU_RELAY.oData[2].7),3));
						ChrCommunication_CAN:= FBRX_BMS_HCU_RELAY.oData[2].3;
						ChrOFFCC2_CAN:= FBRX_BMS_HCU_RELAY.oData[2].2;
						ChrONCC_CAN:= (BIT_TO_BYTE(FBRX_BMS_HCU_RELAY.oData[2].1)+SHL(BIT_TO_BYTE(FBRX_BMS_HCU_RELAY.oData[2].0),1));
						ChrReqVolt_MSB_CAN:=FBRX_BMS_HCU_RELAY.oData[5] + SHL(BYTE_TO_INT(FBRX_BMS_HCU_RELAY.oData[4]),8);
						ChrReqCurr_MSB_CAN:=FBRX_BMS_HCU_RELAY.oData[7] + SHL(BYTE_TO_INT(FBRX_BMS_HCU_RELAY.oData[6]),8);
				ELSIF FBRX_BMS_HCU_RELAY .oCanTimeout THEN										(* If timeout flag is enabled switch off LedRed *)
				 (*Crear los errores necesarios para cuando no se leen las variable despues del time out*)
						Counter_time_out_BATTERY:=Counter_time_out_BATTERY+1;
				END_IF
		FBRX_BMS_HCU_POWER  (	iCAN			:= ADR(GVL.H_CAN_RX_6),  				(* Structure for sending / receiving CAN messages *)
								iCanId				:= 16#186240F3,							(* CAN Id of receiving message *) 
								iCanIdExtended		:= TRUE,  							(* Standard CAN Frame *)
								iTimeoutLimit		:= T#500MS,							(* Timeout after 500ms - Flag will be set *) 
								oByteCount			=> , 
								oData				=> , 
								oNewData			=> , 
								oCanTimeout			=> , 
								oReceiverId			=> , 
								oTooManyReceivers	=> );	
				
								
				IF FBRX_BMS_HCU_POWER   .oNewData THEN											(* If new CAN data is available *)
						
						MaxTemp_CAN:=FBRX_BMS_HCU_POWER.oData[1]+SHL(BYTE_TO_INT(FBRX_BMS_HCU_POWER.oData[0]),8);
						MinTemp_CAN:=FBRX_BMS_HCU_POWER.oData[3]+SHL(BYTE_TO_INT(FBRX_BMS_HCU_POWER.oData[2]),8);
						MaxTempNo_CAN:=FBRX_BMS_HCU_POWER.oData[5]+SHL(BYTE_TO_INT(FBRX_BMS_HCU_POWER.oData[4]),8);
						MinTempNo_CAN:=FBRX_BMS_HCU_POWER.oData[7]+SHL(BYTE_TO_INT(FBRX_BMS_HCU_POWER.oData[6]),8);
						
				ELSIF FBRX_BMS_HCU_POWER .oCanTimeout THEN										(* If timeout flag is enabled switch off LedRed *)
				 (*Crear los errores necesarios para cuando no se leen las variable despues del time out*)
						Counter_time_out_BATTERY:=Counter_time_out_BATTERY+1;
				END_IF
		FBRX_BMS_HCU_ALARM  (	iCAN			:= ADR(GVL.H_CAN_RX_6),  				(* Structure for sending / receiving CAN messages *)
								iCanId				:= 16#186540F3,							(* CAN Id of receiving message *) 
								iCanIdExtended		:= TRUE,  							(* Standard CAN Frame *)
								iTimeoutLimit		:= T#500MS,							(* Timeout after 500ms - Flag will be set *) 
								oByteCount			=> , 
								oData				=> , 
								oNewData			=> , 
								oCanTimeout			=> , 
								oReceiverId			=> , 
								oTooManyReceivers	=> );	
				
								
				IF FBRX_BMS_HCU_POWER   .oNewData THEN											(* If new CAN data is available *)
						
						ALM_CELL_OV_CAN:= (BIT_TO_BYTE(FBRX_BMS_HCU_ALARM.oData[0].6)+SHL(BIT_TO_BYTE(FBRX_BMS_HCU_ALARM.oData[0].7),1));
						ALM_CELL_UV_CAN:= (BIT_TO_BYTE(FBRX_BMS_HCU_ALARM.oData[0].4)+SHL(BIT_TO_BYTE(FBRX_BMS_HCU_ALARM.oData[0].5),1));
						ALM_CELL_OT_CAN:= (BIT_TO_BYTE(FBRX_BMS_HCU_ALARM.oData[0].2)+SHL(BIT_TO_BYTE(FBRX_BMS_HCU_ALARM.oData[0].3),1));
						ALM_CELL_UT_CAN:= (BIT_TO_BYTE(FBRX_BMS_HCU_ALARM.oData[0].1)+SHL(BIT_TO_BYTE(FBRX_BMS_HCU_ALARM.oData[0].0),1));
						
						ALM_CELL_LBK_CAN := FBRX_BMS_HCU_ALARM.oData[1].7;
						ALM_CELL_TBK_CAN := FBRX_BMS_HCU_ALARM.oData[1].6;
						ALM_BATT_DV_CAN:= (BIT_TO_BYTE(FBRX_BMS_HCU_ALARM.oData[1].4)+SHL(BIT_TO_BYTE(FBRX_BMS_HCU_ALARM.oData[1].5),1));
						ALM_BATT_DT_CAN:= (BIT_TO_BYTE(FBRX_BMS_HCU_ALARM.oData[1].2)+SHL(BIT_TO_BYTE(FBRX_BMS_HCU_ALARM.oData[1].3),1));
						ALM_BATT_OV_CAN:= (BIT_TO_BYTE(FBRX_BMS_HCU_ALARM.oData[1].1)+SHL(BIT_TO_BYTE(FBRX_BMS_HCU_ALARM.oData[1].0),1));
						
						ALM_BATT_UV_CAN:= (BIT_TO_BYTE(FBRX_BMS_HCU_ALARM.oData[2].6)+SHL(BIT_TO_BYTE(FBRX_BMS_HCU_ALARM.oData[2].7),1));
						ALM_BATT_OC_CAN:= (BIT_TO_BYTE(FBRX_BMS_HCU_ALARM.oData[2].4)+SHL(BIT_TO_BYTE(FBRX_BMS_HCU_ALARM.oData[2].5),1));
						ALM_BATT_UC_CAN:= (BIT_TO_BYTE(FBRX_BMS_HCU_ALARM.oData[2].2)+SHL(BIT_TO_BYTE(FBRX_BMS_HCU_ALARM.oData[2].3),1));
						ALM_CHRG_OCS_CAN:= (BIT_TO_BYTE(FBRX_BMS_HCU_ALARM.oData[2].1)+SHL(BIT_TO_BYTE(FBRX_BMS_HCU_ALARM.oData[2].0),1));
						
						ALM_DSCH_OCS_CAN:= (BIT_TO_BYTE(FBRX_BMS_HCU_ALARM.oData[3].6)+SHL(BIT_TO_BYTE(FBRX_BMS_HCU_ALARM.oData[3].7),1));
						ALM_CHRG_OCT_CAN:= (BIT_TO_BYTE(FBRX_BMS_HCU_ALARM.oData[3].4)+SHL(BIT_TO_BYTE(FBRX_BMS_HCU_ALARM.oData[3].5),1));
						ALM_DSCH_OCT_CAN:= (BIT_TO_BYTE(FBRX_BMS_HCU_ALARM.oData[3].2)+SHL(BIT_TO_BYTE(FBRX_BMS_HCU_ALARM.oData[3].3),1));
						ALM_BSU_OFFLINE_CAN:= (BIT_TO_BYTE(FBRX_BMS_HCU_ALARM.oData[3].1)+SHL(BIT_TO_BYTE(FBRX_BMS_HCU_ALARM.oData[3].0),1));
						
						ALM_BSU_FAULT_CAN :=  FBRX_BMS_HCU_ALARM.oData[4].7;
						ALM_LEAK_OC_CAN:= (BIT_TO_BYTE(FBRX_BMS_HCU_ALARM.oData[4].5)+SHL(BIT_TO_BYTE(FBRX_BMS_HCU_ALARM.oData[1].6),1));
						ALM_PRECHRG_FAIL_CAN :=  FBRX_BMS_HCU_ALARM.oData[4].4;
						ALM_AUX_FAIL_CAN :=  FBRX_BMS_HCU_ALARM.oData[4].3;
						ALM_BMU_FAIL_CAN :=  FBRX_BMS_HCU_ALARM.oData[4].2;
						ALM_VCU_OFFLINE_CAN:= (BIT_TO_BYTE(FBRX_BMS_HCU_ALARM.oData[4].1)+SHL(BIT_TO_BYTE(FBRX_BMS_HCU_ALARM.oData[4].0),1));
						
						ALM_HVREL_FAIL_CAN := FBRX_BMS_HCU_ALARM.oData[5].7;
						ALM_HALL_BREAK_CAN := FBRX_BMS_HCU_ALARM.oData[5].6;
						
				ELSIF FBRX_BMS_HCU_POWER .oCanTimeout THEN										(* If timeout flag is enabled switch off LedRed *)
				 (*Crear los errores necesarios para cuando no se leen las variable despues del time out*)
						Counter_time_out_BATTERY:=Counter_time_out_BATTERY+1;
				END_IF
		FBRX_BMS_HCU_CELLV_1  (	iCAN			:= ADR(GVL.H_CAN_RX_6),  				(* Structure for sending / receiving CAN messages *)
								iCanId				:= 16#180050F3,							(* CAN Id of receiving message *) 
								iCanIdExtended		:= TRUE,  							(* Standard CAN Frame *)
								iTimeoutLimit		:= T#500MS,							(* Timeout after 500ms - Flag will be set *) 
								oByteCount			=> , 
								oData				=> , 
								oNewData			=> , 
								oCanTimeout			=> , 
								oReceiverId			=> , 
								oTooManyReceivers	=> );	
				
								
				IF FBRX_BMS_HCU_CELLV_1   .oNewData THEN											(* If new CAN data is available *)
						
						CellVoltN_1_CAN:=FBRX_BMS_HCU_CELLV_1.oData[1]+SHL(BYTE_TO_INT(FBRX_BMS_HCU_CELLV_1.oData[0]),8);
						CellVoltN_2_CAN:=FBRX_BMS_HCU_CELLV_1.oData[3]+SHL(BYTE_TO_INT(FBRX_BMS_HCU_CELLV_1.oData[2]),8);
						CellVoltN_3_CAN:=FBRX_BMS_HCU_CELLV_1.oData[5]+SHL(BYTE_TO_INT(FBRX_BMS_HCU_CELLV_1.oData[4]),8);
						CellVoltN_4_CAN:=FBRX_BMS_HCU_CELLV_1.oData[7]+SHL(BYTE_TO_INT(FBRX_BMS_HCU_CELLV_1.oData[6]),8);
					
				ELSIF FBRX_BMS_HCU_CELLV_1 .oCanTimeout THEN										(* If timeout flag is enabled switch off LedRed *)
				 (*Crear los errores necesarios para cuando no se leen las variable despues del time out*)
						Counter_time_out_BATTERY:=Counter_time_out_BATTERY+1;
				END_IF
		FBRX_BMS_HCU_CELLV_2  (	iCAN			:= ADR(GVL.H_CAN_RX_6),  				(* Structure for sending / receiving CAN messages *)
								iCanId				:= 16#180150F3,							(* CAN Id of receiving message *) 
								iCanIdExtended		:= TRUE,  							(* Standard CAN Frame *)
								iTimeoutLimit		:= T#500MS,							(* Timeout after 500ms - Flag will be set *) 
								oByteCount			=> , 
								oData				=> , 
								oNewData			=> , 
								oCanTimeout			=> , 
								oReceiverId			=> , 
								oTooManyReceivers	=> );	
				
								
				IF FBRX_BMS_HCU_CELLV_1   .oNewData THEN											(* If new CAN data is available *)
						
						CellVoltN_5_CAN:=FBRX_BMS_HCU_CELLV_2.oData[1]+SHL(BYTE_TO_INT(FBRX_BMS_HCU_CELLV_2.oData[0]),8);
						CellVoltN_6_CAN:=FBRX_BMS_HCU_CELLV_2.oData[3]+SHL(BYTE_TO_INT(FBRX_BMS_HCU_CELLV_2.oData[2]),8);
						CellVoltN_7_CAN:=FBRX_BMS_HCU_CELLV_2.oData[5]+SHL(BYTE_TO_INT(FBRX_BMS_HCU_CELLV_2.oData[4]),8);
						CellVoltN_8_CAN:=FBRX_BMS_HCU_CELLV_2.oData[7]+SHL(BYTE_TO_INT(FBRX_BMS_HCU_CELLV_2.oData[6]),8);
					
				ELSIF FBRX_BMS_HCU_CELLV_2 .oCanTimeout THEN										(* If timeout flag is enabled switch off LedRed *)
				 (*Crear los errores necesarios para cuando no se leen las variable despues del time out*)
						Counter_time_out_BATTERY:=Counter_time_out_BATTERY+1;
				END_IF
		FBRX_BMS_HCU_CELLV_3  (	iCAN			:= ADR(GVL.H_CAN_RX_6),  				(* Structure for sending / receiving CAN messages *)
								iCanId				:= 16#180250F3,							(* CAN Id of receiving message *) 
								iCanIdExtended		:= TRUE,  							(* Standard CAN Frame *)
								iTimeoutLimit		:= T#500MS,							(* Timeout after 500ms - Flag will be set *) 
								oByteCount			=> , 
								oData				=> , 
								oNewData			=> , 
								oCanTimeout			=> , 
								oReceiverId			=> , 
								oTooManyReceivers	=> );	
				
								
				IF FBRX_BMS_HCU_CELLV_3   .oNewData THEN											(* If new CAN data is available *)
						
						CellVoltN_9_CAN:=FBRX_BMS_HCU_CELLV_3.oData[1]+SHL(BYTE_TO_INT(FBRX_BMS_HCU_CELLV_3.oData[0]),8);
						CellVoltN_10_CAN:=FBRX_BMS_HCU_CELLV_3.oData[3]+SHL(BYTE_TO_INT(FBRX_BMS_HCU_CELLV_3.oData[2]),8);
						CellVoltN_11_CAN:=FBRX_BMS_HCU_CELLV_3.oData[5]+SHL(BYTE_TO_INT(FBRX_BMS_HCU_CELLV_3.oData[4]),8);
						CellVoltN_12_CAN:=FBRX_BMS_HCU_CELLV_3.oData[7]+SHL(BYTE_TO_INT(FBRX_BMS_HCU_CELLV_3.oData[6]),8);
					
				ELSIF FBRX_BMS_HCU_CELLV_3 .oCanTimeout THEN										(* If timeout flag is enabled switch off LedRed *)
				 (*Crear los errores necesarios para cuando no se leen las variable despues del time out*)
						Counter_time_out_BATTERY:=Counter_time_out_BATTERY+1;
				END_IF
		FBRX_BMS_HCU_CELLV_4  (	iCAN			:= ADR(GVL.H_CAN_RX_6),  				(* Structure for sending / receiving CAN messages *)
								iCanId				:= 16#180350F3,							(* CAN Id of receiving message *) 
								iCanIdExtended		:= TRUE,  							(* Standard CAN Frame *)
								iTimeoutLimit		:= T#500MS,							(* Timeout after 500ms - Flag will be set *) 
								oByteCount			=> , 
								oData				=> , 
								oNewData			=> , 
								oCanTimeout			=> , 
								oReceiverId			=> , 
								oTooManyReceivers	=> );	
				
								
				IF FBRX_BMS_HCU_CELLV_4   .oNewData THEN											(* If new CAN data is available *)
						
						CellVoltN_13_CAN:=FBRX_BMS_HCU_CELLV_4.oData[1]+SHL(BYTE_TO_INT(FBRX_BMS_HCU_CELLV_4.oData[0]),8);
						CellVoltN_14_CAN:=FBRX_BMS_HCU_CELLV_4.oData[3]+SHL(BYTE_TO_INT(FBRX_BMS_HCU_CELLV_4.oData[2]),8);
						CellVoltN_15_CAN:=FBRX_BMS_HCU_CELLV_4.oData[5]+SHL(BYTE_TO_INT(FBRX_BMS_HCU_CELLV_4.oData[4]),8);
						CellVoltN_16_CAN:=FBRX_BMS_HCU_CELLV_4.oData[7]+SHL(BYTE_TO_INT(FBRX_BMS_HCU_CELLV_4.oData[6]),8);
					
				ELSIF FBRX_BMS_HCU_CELLV_4 .oCanTimeout THEN										(* If timeout flag is enabled switch off LedRed *)
				 (*Crear los errores necesarios para cuando no se leen las variable despues del time out*)
						Counter_time_out_BATTERY:=Counter_time_out_BATTERY+1;
				END_IF
		FBRX_BMS_HCU_CELLV_5  (	iCAN			:= ADR(GVL.H_CAN_RX_6),  				(* Structure for sending / receiving CAN messages *)
								iCanId				:= 16#180450F3,							(* CAN Id of receiving message *) 
								iCanIdExtended		:= TRUE,  							(* Standard CAN Frame *)
								iTimeoutLimit		:= T#500MS,							(* Timeout after 500ms - Flag will be set *) 
								oByteCount			=> , 
								oData				=> , 
								oNewData			=> , 
								oCanTimeout			=> , 
								oReceiverId			=> , 
								oTooManyReceivers	=> );	
				
								
				IF FBRX_BMS_HCU_CELLV_1   .oNewData THEN											(* If new CAN data is available *)
						
						CellVoltN_17_CAN:=FBRX_BMS_HCU_CELLV_5.oData[1]+SHL(BYTE_TO_INT(FBRX_BMS_HCU_CELLV_5.oData[0]),8);
						CellVoltN_18_CAN:=FBRX_BMS_HCU_CELLV_5.oData[3]+SHL(BYTE_TO_INT(FBRX_BMS_HCU_CELLV_5.oData[2]),8);
						CellVoltN_19_CAN:=FBRX_BMS_HCU_CELLV_5.oData[5]+SHL(BYTE_TO_INT(FBRX_BMS_HCU_CELLV_5.oData[4]),8);
						CellVoltN_20_CAN:=FBRX_BMS_HCU_CELLV_5.oData[7]+SHL(BYTE_TO_INT(FBRX_BMS_HCU_CELLV_5.oData[6]),8);
					
				ELSIF FBRX_BMS_HCU_CELLV_5 .oCanTimeout THEN										(* If timeout flag is enabled switch off LedRed *)
				 (*Crear los errores necesarios para cuando no se leen las variable despues del time out*)
						Counter_time_out_BATTERY:=Counter_time_out_BATTERY+1;
				END_IF
		FBRX_BMS_HCU_CELLV_6  (	iCAN			:= ADR(GVL.H_CAN_RX_6),  				(* Structure for sending / receiving CAN messages *)
								iCanId				:= 16#180550F3,							(* CAN Id of receiving message *) 
								iCanIdExtended		:= TRUE,  							(* Standard CAN Frame *)
								iTimeoutLimit		:= T#500MS,							(* Timeout after 500ms - Flag will be set *) 
								oByteCount			=> , 
								oData				=> , 
								oNewData			=> , 
								oCanTimeout			=> , 
								oReceiverId			=> , 
								oTooManyReceivers	=> );	
				
								
				IF FBRX_BMS_HCU_CELLV_6   .oNewData THEN											(* If new CAN data is available *)
						
						CellVoltN_21_CAN:=FBRX_BMS_HCU_CELLV_6.oData[1]+SHL(BYTE_TO_INT(FBRX_BMS_HCU_CELLV_6.oData[0]),8);
						CellVoltN_22_CAN:=FBRX_BMS_HCU_CELLV_6.oData[3]+SHL(BYTE_TO_INT(FBRX_BMS_HCU_CELLV_6.oData[2]),8);
						CellVoltN_23_CAN:=FBRX_BMS_HCU_CELLV_6.oData[5]+SHL(BYTE_TO_INT(FBRX_BMS_HCU_CELLV_6.oData[4]),8);
						CellVoltN_24_CAN:=FBRX_BMS_HCU_CELLV_6.oData[7]+SHL(BYTE_TO_INT(FBRX_BMS_HCU_CELLV_6.oData[6]),8);
					
				ELSIF FBRX_BMS_HCU_CELLV_6 .oCanTimeout THEN										(* If timeout flag is enabled switch off LedRed *)
				 (*Crear los errores necesarios para cuando no se leen las variable despues del time out*)
						Counter_time_out_BATTERY:=Counter_time_out_BATTERY+1;
				END_IF
		FBRX_BMS_HCU_CELLV_7  (	iCAN			:= ADR(GVL.H_CAN_RX_6),  				(* Structure for sending / receiving CAN messages *)
								iCanId				:= 16#180650F3,							(* CAN Id of receiving message *) 
								iCanIdExtended		:= TRUE,  							(* Standard CAN Frame *)
								iTimeoutLimit		:= T#500MS,							(* Timeout after 500ms - Flag will be set *) 
								oByteCount			=> , 
								oData				=> , 
								oNewData			=> , 
								oCanTimeout			=> , 
								oReceiverId			=> , 
								oTooManyReceivers	=> );	
				
								
				IF FBRX_BMS_HCU_CELLV_7   .oNewData THEN											(* If new CAN data is available *)
						
						CellVoltN_25_CAN:=FBRX_BMS_HCU_CELLV_7.oData[1]+SHL(BYTE_TO_INT(FBRX_BMS_HCU_CELLV_7.oData[0]),8);
						CellVoltN_26_CAN:=FBRX_BMS_HCU_CELLV_7.oData[3]+SHL(BYTE_TO_INT(FBRX_BMS_HCU_CELLV_7.oData[2]),8);
						CellVoltN_27_CAN:=FBRX_BMS_HCU_CELLV_7.oData[5]+SHL(BYTE_TO_INT(FBRX_BMS_HCU_CELLV_7.oData[4]),8);
						CellVoltN_28_CAN:=FBRX_BMS_HCU_CELLV_7.oData[7]+SHL(BYTE_TO_INT(FBRX_BMS_HCU_CELLV_7.oData[6]),8);
					
				ELSIF FBRX_BMS_HCU_CELLV_7 .oCanTimeout THEN										(* If timeout flag is enabled switch off LedRed *)
				 (*Crear los errores necesarios para cuando no se leen las variable despues del time out*)
						Counter_time_out_BATTERY:=Counter_time_out_BATTERY+1;
				END_IF
		FBRX_BMS_HCU_CELLV_8  (	iCAN			:= ADR(GVL.H_CAN_RX_6),  				(* Structure for sending / receiving CAN messages *)
								iCanId				:= 16#180750F3,							(* CAN Id of receiving message *) 
								iCanIdExtended		:= TRUE,  							(* Standard CAN Frame *)
								iTimeoutLimit		:= T#500MS,							(* Timeout after 500ms - Flag will be set *) 
								oByteCount			=> , 
								oData				=> , 
								oNewData			=> , 
								oCanTimeout			=> , 
								oReceiverId			=> , 
								oTooManyReceivers	=> );	
				
								
				IF FBRX_BMS_HCU_CELLV_8   .oNewData THEN											(* If new CAN data is available *)
						
						CellVoltN_29_CAN:=FBRX_BMS_HCU_CELLV_8.oData[1]+SHL(BYTE_TO_INT(FBRX_BMS_HCU_CELLV_8.oData[0]),8);
						CellVoltN_30_CAN:=FBRX_BMS_HCU_CELLV_8.oData[3]+SHL(BYTE_TO_INT(FBRX_BMS_HCU_CELLV_8.oData[2]),8);
						CellVoltN_31_CAN:=FBRX_BMS_HCU_CELLV_8.oData[5]+SHL(BYTE_TO_INT(FBRX_BMS_HCU_CELLV_8.oData[4]),8);
						CellVoltN_32_CAN:=FBRX_BMS_HCU_CELLV_8.oData[7]+SHL(BYTE_TO_INT(FBRX_BMS_HCU_CELLV_8.oData[6]),8);
					
				ELSIF FBRX_BMS_HCU_CELLV_8 .oCanTimeout THEN										(* If timeout flag is enabled switch off LedRed *)
				 (*Crear los errores necesarios para cuando no se leen las variable despues del time out*)
						Counter_time_out_BATTERY:=Counter_time_out_BATTERY+1;
				END_IF
		FBRX_BMS_HCU_CELLV_9  (	iCAN			:= ADR(GVL.H_CAN_RX_6),  				(* Structure for sending / receiving CAN messages *)
								iCanId				:= 16#180850F3,							(* CAN Id of receiving message *) 
								iCanIdExtended		:= TRUE,  							(* Standard CAN Frame *)
								iTimeoutLimit		:= T#500MS,							(* Timeout after 500ms - Flag will be set *) 
								oByteCount			=> , 
								oData				=> , 
								oNewData			=> , 
								oCanTimeout			=> , 
								oReceiverId			=> , 
								oTooManyReceivers	=> );	
				
								
				IF FBRX_BMS_HCU_CELLV_9   .oNewData THEN											(* If new CAN data is available *)
						
						CellVoltN_33_CAN:=FBRX_BMS_HCU_CELLV_9.oData[1]+SHL(BYTE_TO_INT(FBRX_BMS_HCU_CELLV_9.oData[0]),8);
						CellVoltN_34_CAN:=FBRX_BMS_HCU_CELLV_9.oData[3]+SHL(BYTE_TO_INT(FBRX_BMS_HCU_CELLV_9.oData[2]),8);
						CellVoltN_35_CAN:=FBRX_BMS_HCU_CELLV_9.oData[5]+SHL(BYTE_TO_INT(FBRX_BMS_HCU_CELLV_9.oData[4]),8);
						CellVoltN_36_CAN:=FBRX_BMS_HCU_CELLV_9.oData[7]+SHL(BYTE_TO_INT(FBRX_BMS_HCU_CELLV_9.oData[6]),8);
					
				ELSIF FBRX_BMS_HCU_CELLV_9 .oCanTimeout THEN										(* If timeout flag is enabled switch off LedRed *)
				 (*Crear los errores necesarios para cuando no se leen las variable despues del time out*)
						Counter_time_out_BATTERY:=Counter_time_out_BATTERY+1;
				END_IF
		FBRX_BMS_HCU_CELLV_10  (	iCAN			:= ADR(GVL.H_CAN_RX_6),  				(* Structure for sending / receiving CAN messages *)
								iCanId				:= 16#180950F3,							(* CAN Id of receiving message *) 
								iCanIdExtended		:= TRUE,  							(* Standard CAN Frame *)
								iTimeoutLimit		:= T#500MS,							(* Timeout after 500ms - Flag will be set *) 
								oByteCount			=> , 
								oData				=> , 
								oNewData			=> , 
								oCanTimeout			=> , 
								oReceiverId			=> , 
								oTooManyReceivers	=> );	
				
								
				IF FBRX_BMS_HCU_CELLV_10   .oNewData THEN											(* If new CAN data is available *)
						
						CellVoltN_37_CAN:=FBRX_BMS_HCU_CELLV_10.oData[1]+SHL(BYTE_TO_INT(FBRX_BMS_HCU_CELLV_10.oData[0]),8);
						CellVoltN_38_CAN:=FBRX_BMS_HCU_CELLV_10.oData[3]+SHL(BYTE_TO_INT(FBRX_BMS_HCU_CELLV_10.oData[2]),8);
						CellVoltN_39_CAN:=FBRX_BMS_HCU_CELLV_10.oData[5]+SHL(BYTE_TO_INT(FBRX_BMS_HCU_CELLV_10.oData[4]),8);
						CellVoltN_40_CAN:=FBRX_BMS_HCU_CELLV_10.oData[7]+SHL(BYTE_TO_INT(FBRX_BMS_HCU_CELLV_10.oData[6]),8);
					
				ELSIF FBRX_BMS_HCU_CELLV_10 .oCanTimeout THEN										(* If timeout flag is enabled switch off LedRed *)
				 (*Crear los errores necesarios para cuando no se leen las variable despues del time out*)
						Counter_time_out_BATTERY:=Counter_time_out_BATTERY+1;
				END_IF
		FBRX_BMS_HCU_CELLV_11  (	iCAN			:= ADR(GVL.H_CAN_RX_6),  				(* Structure for sending / receiving CAN messages *)
								iCanId				:= 16#180A50F3,							(* CAN Id of receiving message *) 
								iCanIdExtended		:= TRUE,  							(* Standard CAN Frame *)
								iTimeoutLimit		:= T#500MS,							(* Timeout after 500ms - Flag will be set *) 
								oByteCount			=> , 
								oData				=> , 
								oNewData			=> , 
								oCanTimeout			=> , 
								oReceiverId			=> , 
								oTooManyReceivers	=> );	
				
								
				IF FBRX_BMS_HCU_CELLV_11   .oNewData THEN											(* If new CAN data is available *)
						
						CellVoltN_41_CAN:=FBRX_BMS_HCU_CELLV_11.oData[1]+SHL(BYTE_TO_INT(FBRX_BMS_HCU_CELLV_11.oData[0]),8);
						CellVoltN_42_CAN:=FBRX_BMS_HCU_CELLV_11.oData[3]+SHL(BYTE_TO_INT(FBRX_BMS_HCU_CELLV_11.oData[2]),8);
						CellVoltN_43_CAN:=FBRX_BMS_HCU_CELLV_11.oData[5]+SHL(BYTE_TO_INT(FBRX_BMS_HCU_CELLV_11.oData[4]),8);
						CellVoltN_44_CAN:=FBRX_BMS_HCU_CELLV_11.oData[7]+SHL(BYTE_TO_INT(FBRX_BMS_HCU_CELLV_11.oData[6]),8);
					
				ELSIF FBRX_BMS_HCU_CELLV_11 .oCanTimeout THEN										(* If timeout flag is enabled switch off LedRed *)
				 (*Crear los errores necesarios para cuando no se leen las variable despues del time out*)
						Counter_time_out_BATTERY:=Counter_time_out_BATTERY+1;
				END_IF
		FBRX_BMS_HCU_CELLV_12  (	iCAN			:= ADR(GVL.H_CAN_RX_6),  				(* Structure for sending / receiving CAN messages *)
								iCanId				:= 16#180B50F3,							(* CAN Id of receiving message *) 
								iCanIdExtended		:= TRUE,  							(* Standard CAN Frame *)
								iTimeoutLimit		:= T#500MS,							(* Timeout after 500ms - Flag will be set *) 
								oByteCount			=> , 
								oData				=> , 
								oNewData			=> , 
								oCanTimeout			=> , 
								oReceiverId			=> , 
								oTooManyReceivers	=> );	
				
								
				IF FBRX_BMS_HCU_CELLV_12   .oNewData THEN											(* If new CAN data is available *)
						
						CellVoltN_45_CAN:=FBRX_BMS_HCU_CELLV_12.oData[1]+SHL(BYTE_TO_INT(FBRX_BMS_HCU_CELLV_12.oData[0]),8);
						CellVoltN_46_CAN:=FBRX_BMS_HCU_CELLV_12.oData[3]+SHL(BYTE_TO_INT(FBRX_BMS_HCU_CELLV_12.oData[2]),8);
						CellVoltN_47_CAN:=FBRX_BMS_HCU_CELLV_12.oData[5]+SHL(BYTE_TO_INT(FBRX_BMS_HCU_CELLV_12.oData[4]),8);
						CellVoltN_48_CAN:=FBRX_BMS_HCU_CELLV_12.oData[7]+SHL(BYTE_TO_INT(FBRX_BMS_HCU_CELLV_12.oData[6]),8);
					
				ELSIF FBRX_BMS_HCU_CELLV_12 .oCanTimeout THEN										(* If timeout flag is enabled switch off LedRed *)
				 (*Crear los errores necesarios para cuando no se leen las variable despues del time out*)
						Counter_time_out_BATTERY:=Counter_time_out_BATTERY+1;
				END_IF
		FBRX_BMS_HCU_CELLV_13  (	iCAN			:= ADR(GVL.H_CAN_RX_6),  				(* Structure for sending / receiving CAN messages *)
								iCanId				:= 16#180C50F3,							(* CAN Id of receiving message *) 
								iCanIdExtended		:= TRUE,  							(* Standard CAN Frame *)
								iTimeoutLimit		:= T#500MS,							(* Timeout after 500ms - Flag will be set *) 
								oByteCount			=> , 
								oData				=> , 
								oNewData			=> , 
								oCanTimeout			=> , 
								oReceiverId			=> , 
								oTooManyReceivers	=> );	
				
								
				IF FBRX_BMS_HCU_CELLV_13   .oNewData THEN											(* If new CAN data is available *)
						
						CellVoltN_49_CAN:=FBRX_BMS_HCU_CELLV_13.oData[1]+SHL(BYTE_TO_INT(FBRX_BMS_HCU_CELLV_13.oData[0]),8);
						CellVoltN_50_CAN:=FBRX_BMS_HCU_CELLV_13.oData[3]+SHL(BYTE_TO_INT(FBRX_BMS_HCU_CELLV_13.oData[2]),8);
						CellVoltN_51_CAN:=FBRX_BMS_HCU_CELLV_13.oData[5]+SHL(BYTE_TO_INT(FBRX_BMS_HCU_CELLV_13.oData[4]),8);
						CellVoltN_52_CAN:=FBRX_BMS_HCU_CELLV_13.oData[7]+SHL(BYTE_TO_INT(FBRX_BMS_HCU_CELLV_13.oData[6]),8);
					
				ELSIF FBRX_BMS_HCU_CELLV_13 .oCanTimeout THEN										(* If timeout flag is enabled switch off LedRed *)
				 (*Crear los errores necesarios para cuando no se leen las variable despues del time out*)
						Counter_time_out_BATTERY:=Counter_time_out_BATTERY+1;
				END_IF
		FBRX_BMS_HCU_CELLV_14  (	iCAN			:= ADR(GVL.H_CAN_RX_6),  				(* Structure for sending / receiving CAN messages *)
								iCanId				:= 16#180D50F3,							(* CAN Id of receiving message *) 
								iCanIdExtended		:= TRUE,  							(* Standard CAN Frame *)
								iTimeoutLimit		:= T#500MS,							(* Timeout after 500ms - Flag will be set *) 
								oByteCount			=> , 
								oData				=> , 
								oNewData			=> , 
								oCanTimeout			=> , 
								oReceiverId			=> , 
								oTooManyReceivers	=> );	
				
								
				IF FBRX_BMS_HCU_CELLV_14   .oNewData THEN											(* If new CAN data is available *)
						
						CellVoltN_53_CAN:=FBRX_BMS_HCU_CELLV_14.oData[1]+SHL(BYTE_TO_INT(FBRX_BMS_HCU_CELLV_14.oData[0]),8);
						CellVoltN_54_CAN:=FBRX_BMS_HCU_CELLV_14.oData[3]+SHL(BYTE_TO_INT(FBRX_BMS_HCU_CELLV_14.oData[2]),8);
						CellVoltN_55_CAN:=FBRX_BMS_HCU_CELLV_14.oData[5]+SHL(BYTE_TO_INT(FBRX_BMS_HCU_CELLV_14.oData[4]),8);
						CellVoltN_56_CAN:=FBRX_BMS_HCU_CELLV_14.oData[7]+SHL(BYTE_TO_INT(FBRX_BMS_HCU_CELLV_14.oData[6]),8);
					
				ELSIF FBRX_BMS_HCU_CELLV_14 .oCanTimeout THEN										(* If timeout flag is enabled switch off LedRed *)
				 (*Crear los errores necesarios para cuando no se leen las variable despues del time out*)
						Counter_time_out_BATTERY:=Counter_time_out_BATTERY+1;
				END_IF
		FBRX_BMS_HCU_CELLV_15  (	iCAN			:= ADR(GVL.H_CAN_RX_6),  				(* Structure for sending / receiving CAN messages *)
								iCanId				:= 16#180E50F3,							(* CAN Id of receiving message *) 
								iCanIdExtended		:= TRUE,  							(* Standard CAN Frame *)
								iTimeoutLimit		:= T#500MS,							(* Timeout after 500ms - Flag will be set *) 
								oByteCount			=> , 
								oData				=> , 
								oNewData			=> , 
								oCanTimeout			=> , 
								oReceiverId			=> , 
								oTooManyReceivers	=> );	
				
								
				IF FBRX_BMS_HCU_CELLV_15   .oNewData THEN											(* If new CAN data is available *)
						
						CellVoltN_57_CAN:=FBRX_BMS_HCU_CELLV_15.oData[1]+SHL(BYTE_TO_INT(FBRX_BMS_HCU_CELLV_15.oData[0]),8);
						CellVoltN_58_CAN:=FBRX_BMS_HCU_CELLV_15.oData[3]+SHL(BYTE_TO_INT(FBRX_BMS_HCU_CELLV_15.oData[2]),8);
						CellVoltN_59_CAN:=FBRX_BMS_HCU_CELLV_15.oData[5]+SHL(BYTE_TO_INT(FBRX_BMS_HCU_CELLV_15.oData[4]),8);
						CellVoltN_60_CAN:=FBRX_BMS_HCU_CELLV_15.oData[7]+SHL(BYTE_TO_INT(FBRX_BMS_HCU_CELLV_15.oData[6]),8);
					
				ELSIF FBRX_BMS_HCU_CELLV_15 .oCanTimeout THEN										(* If timeout flag is enabled switch off LedRed *)
				 (*Crear los errores necesarios para cuando no se leen las variable despues del time out*)
						Counter_time_out_BATTERY:=Counter_time_out_BATTERY+1;
				END_IF
		FBRX_BMS_HCU_CELLV_16  (	iCAN			:= ADR(GVL.H_CAN_RX_6),  				(* Structure for sending / receiving CAN messages *)
								iCanId				:= 16#180F50F3,							(* CAN Id of receiving message *) 
								iCanIdExtended		:= TRUE,  							(* Standard CAN Frame *)
								iTimeoutLimit		:= T#500MS,							(* Timeout after 500ms - Flag will be set *) 
								oByteCount			=> , 
								oData				=> , 
								oNewData			=> , 
								oCanTimeout			=> , 
								oReceiverId			=> , 
								oTooManyReceivers	=> );	
				
								
				IF FBRX_BMS_HCU_CELLV_16   .oNewData THEN											(* If new CAN data is available *)
						
						CellVoltN_61_CAN:=FBRX_BMS_HCU_CELLV_16.oData[1]+SHL(BYTE_TO_INT(FBRX_BMS_HCU_CELLV_17.oData[0]),8);
						CellVoltN_62_CAN:=FBRX_BMS_HCU_CELLV_16.oData[3]+SHL(BYTE_TO_INT(FBRX_BMS_HCU_CELLV_17.oData[2]),8);
						CellVoltN_63_CAN:=FBRX_BMS_HCU_CELLV_16.oData[5]+SHL(BYTE_TO_INT(FBRX_BMS_HCU_CELLV_17.oData[4]),8);
						CellVoltN_64_CAN:=FBRX_BMS_HCU_CELLV_16.oData[7]+SHL(BYTE_TO_INT(FBRX_BMS_HCU_CELLV_17.oData[6]),8);
					
				ELSIF FBRX_BMS_HCU_CELLV_17 .oCanTimeout THEN										(* If timeout flag is enabled switch off LedRed *)
				 (*Crear los errores necesarios para cuando no se leen las variable despues del time out*)
						Counter_time_out_BATTERY:=Counter_time_out_BATTERY+1;
				END_IF
		FBRX_BMS_HCU_CELLV_17  (	iCAN			:= ADR(GVL.H_CAN_RX_6),  				(* Structure for sending / receiving CAN messages *)
								iCanId				:= 16#181050F3,							(* CAN Id of receiving message *) 
								iCanIdExtended		:= TRUE,  							(* Standard CAN Frame *)
								iTimeoutLimit		:= T#500MS,							(* Timeout after 500ms - Flag will be set *) 
								oByteCount			=> , 
								oData				=> , 
								oNewData			=> , 
								oCanTimeout			=> , 
								oReceiverId			=> , 
								oTooManyReceivers	=> );	
				
								
				IF FBRX_BMS_HCU_CELLV_17   .oNewData THEN											(* If new CAN data is available *)
						
						CellVoltN_65_CAN:=FBRX_BMS_HCU_CELLV_17.oData[1]+SHL(BYTE_TO_INT(FBRX_BMS_HCU_CELLV_17.oData[0]),8);
						CellVoltN_66_CAN:=FBRX_BMS_HCU_CELLV_17.oData[3]+SHL(BYTE_TO_INT(FBRX_BMS_HCU_CELLV_17.oData[2]),8);
						CellVoltN_67_CAN:=FBRX_BMS_HCU_CELLV_17.oData[5]+SHL(BYTE_TO_INT(FBRX_BMS_HCU_CELLV_17.oData[4]),8);
						CellVoltN_68_CAN:=FBRX_BMS_HCU_CELLV_17.oData[7]+SHL(BYTE_TO_INT(FBRX_BMS_HCU_CELLV_17.oData[6]),8);
					
				ELSIF FBRX_BMS_HCU_CELLV_17 .oCanTimeout THEN										(* If timeout flag is enabled switch off LedRed *)
				 (*Crear los errores necesarios para cuando no se leen las variable despues del time out*)
						Counter_time_out_BATTERY:=Counter_time_out_BATTERY+1;
				END_IF
		FBRX_BMS_HCU_CELLV_18  (	iCAN			:= ADR(GVL.H_CAN_RX_6),  				(* Structure for sending / receiving CAN messages *)
								iCanId				:= 16#181150F3,							(* CAN Id of receiving message *) 
								iCanIdExtended		:= TRUE,  							(* Standard CAN Frame *)
								iTimeoutLimit		:= T#500MS,							(* Timeout after 500ms - Flag will be set *) 
								oByteCount			=> , 
								oData				=> , 
								oNewData			=> , 
								oCanTimeout			=> , 
								oReceiverId			=> , 
								oTooManyReceivers	=> );	
				
								
				IF FBRX_BMS_HCU_CELLV_18   .oNewData THEN											(* If new CAN data is available *)
						
						CellVoltN_69_CAN:=FBRX_BMS_HCU_CELLV_18.oData[1]+SHL(BYTE_TO_INT(FBRX_BMS_HCU_CELLV_18.oData[0]),8);
						CellVoltN_70_CAN:=FBRX_BMS_HCU_CELLV_18.oData[3]+SHL(BYTE_TO_INT(FBRX_BMS_HCU_CELLV_18.oData[2]),8);
						CellVoltN_71_CAN:=FBRX_BMS_HCU_CELLV_18.oData[5]+SHL(BYTE_TO_INT(FBRX_BMS_HCU_CELLV_18.oData[4]),8);
						CellVoltN_72_CAN:=FBRX_BMS_HCU_CELLV_18.oData[7]+SHL(BYTE_TO_INT(FBRX_BMS_HCU_CELLV_18.oData[6]),8);
					
				ELSIF FBRX_BMS_HCU_CELLV_18 .oCanTimeout THEN										(* If timeout flag is enabled switch off LedRed *)
				 (*Crear los errores necesarios para cuando no se leen las variable despues del time out*)
						Counter_time_out_BATTERY:=Counter_time_out_BATTERY+1;
				END_IF
		FBRX_BMS_HCU_CELLV_19  (	iCAN			:= ADR(GVL.H_CAN_RX_6),  				(* Structure for sending / receiving CAN messages *)
								iCanId				:= 16#181250F3,							(* CAN Id of receiving message *) 
								iCanIdExtended		:= TRUE,  							(* Standard CAN Frame *)
								iTimeoutLimit		:= T#500MS,							(* Timeout after 500ms - Flag will be set *) 
								oByteCount			=> , 
								oData				=> , 
								oNewData			=> , 
								oCanTimeout			=> , 
								oReceiverId			=> , 
								oTooManyReceivers	=> );	
				
								
				IF FBRX_BMS_HCU_CELLV_19   .oNewData THEN											(* If new CAN data is available *)
						
						CellVoltN_73_CAN:=FBRX_BMS_HCU_CELLV_19.oData[1]+SHL(BYTE_TO_INT(FBRX_BMS_HCU_CELLV_19.oData[0]),8);
						CellVoltN_74_CAN:=FBRX_BMS_HCU_CELLV_19.oData[3]+SHL(BYTE_TO_INT(FBRX_BMS_HCU_CELLV_19.oData[2]),8);
						CellVoltN_75_CAN:=FBRX_BMS_HCU_CELLV_19.oData[5]+SHL(BYTE_TO_INT(FBRX_BMS_HCU_CELLV_19.oData[4]),8);
						CellVoltN_76_CAN:=FBRX_BMS_HCU_CELLV_19.oData[7]+SHL(BYTE_TO_INT(FBRX_BMS_HCU_CELLV_19.oData[6]),8);
					
				ELSIF FBRX_BMS_HCU_CELLV_19 .oCanTimeout THEN										(* If timeout flag is enabled switch off LedRed *)
				 (*Crear los errores necesarios para cuando no se leen las variable despues del time out*)
						Counter_time_out_BATTERY:=Counter_time_out_BATTERY+1;
				END_IF
		FBRX_BMS_HCU_CELLV_20  (	iCAN			:= ADR(GVL.H_CAN_RX_6),  				(* Structure for sending / receiving CAN messages *)
								iCanId				:= 16#181350F3,							(* CAN Id of receiving message *) 
								iCanIdExtended		:= TRUE,  							(* Standard CAN Frame *)
								iTimeoutLimit		:= T#500MS,							(* Timeout after 500ms - Flag will be set *) 
								oByteCount			=> , 
								oData				=> , 
								oNewData			=> , 
								oCanTimeout			=> , 
								oReceiverId			=> , 
								oTooManyReceivers	=> );	
				
								
				IF FBRX_BMS_HCU_CELLV_20   .oNewData THEN											(* If new CAN data is available *)
						
						CellVoltN_77_CAN:=FBRX_BMS_HCU_CELLV_20.oData[1]+SHL(BYTE_TO_INT(FBRX_BMS_HCU_CELLV_20.oData[0]),8);
						CellVoltN_78_CAN:=FBRX_BMS_HCU_CELLV_20.oData[3]+SHL(BYTE_TO_INT(FBRX_BMS_HCU_CELLV_20.oData[2]),8);
						CellVoltN_79_CAN:=FBRX_BMS_HCU_CELLV_20.oData[5]+SHL(BYTE_TO_INT(FBRX_BMS_HCU_CELLV_20.oData[4]),8);
						CellVoltN_80_CAN:=FBRX_BMS_HCU_CELLV_20.oData[7]+SHL(BYTE_TO_INT(FBRX_BMS_HCU_CELLV_20.oData[6]),8);
					
				ELSIF FBRX_BMS_HCU_CELLV_20 .oCanTimeout THEN										(* If timeout flag is enabled switch off LedRed *)
				 (*Crear los errores necesarios para cuando no se leen las variable despues del time out*)
						Counter_time_out_BATTERY:=Counter_time_out_BATTERY+1;
				END_IF
		FBRX_BMS_HCU_CELLV_21  (	iCAN			:= ADR(GVL.H_CAN_RX_6),  				(* Structure for sending / receiving CAN messages *)
								iCanId				:= 16#181450F3,							(* CAN Id of receiving message *) 
								iCanIdExtended		:= TRUE,  							(* Standard CAN Frame *)
								iTimeoutLimit		:= T#500MS,							(* Timeout after 500ms - Flag will be set *) 
								oByteCount			=> , 
								oData				=> , 
								oNewData			=> , 
								oCanTimeout			=> , 
								oReceiverId			=> , 
								oTooManyReceivers	=> );	
				
								
				IF FBRX_BMS_HCU_CELLV_21   .oNewData THEN											(* If new CAN data is available *)
						
						CellVoltN_81_CAN:=FBRX_BMS_HCU_CELLV_21.oData[1]+SHL(BYTE_TO_INT(FBRX_BMS_HCU_CELLV_21.oData[0]),8);
						CellVoltN_82_CAN:=FBRX_BMS_HCU_CELLV_21.oData[3]+SHL(BYTE_TO_INT(FBRX_BMS_HCU_CELLV_21.oData[2]),8);
						CellVoltN_83_CAN:=FBRX_BMS_HCU_CELLV_21.oData[5]+SHL(BYTE_TO_INT(FBRX_BMS_HCU_CELLV_21.oData[4]),8);
						CellVoltN_84_CAN:=FBRX_BMS_HCU_CELLV_21.oData[7]+SHL(BYTE_TO_INT(FBRX_BMS_HCU_CELLV_21.oData[6]),8);
					
				ELSIF FBRX_BMS_HCU_CELLV_21 .oCanTimeout THEN										(* If timeout flag is enabled switch off LedRed *)
				 (*Crear los errores necesarios para cuando no se leen las variable despues del time out*)
						Counter_time_out_BATTERY:=Counter_time_out_BATTERY+1;
				END_IF
		FBRX_BMS_HCU_CELLV_22  (	iCAN			:= ADR(GVL.H_CAN_RX_6),  				(* Structure for sending / receiving CAN messages *)
								iCanId				:= 16#181550F3,							(* CAN Id of receiving message *) 
								iCanIdExtended		:= TRUE,  							(* Standard CAN Frame *)
								iTimeoutLimit		:= T#500MS,							(* Timeout after 500ms - Flag will be set *) 
								oByteCount			=> , 
								oData				=> , 
								oNewData			=> , 
								oCanTimeout			=> , 
								oReceiverId			=> , 
								oTooManyReceivers	=> );	
				
								
				IF FBRX_BMS_HCU_CELLV_22   .oNewData THEN											(* If new CAN data is available *)
						
						CellVoltN_85_CAN:=FBRX_BMS_HCU_CELLV_22.oData[1]+SHL(BYTE_TO_INT(FBRX_BMS_HCU_CELLV_22.oData[0]),8);
						CellVoltN_86_CAN:=FBRX_BMS_HCU_CELLV_22.oData[3]+SHL(BYTE_TO_INT(FBRX_BMS_HCU_CELLV_22.oData[2]),8);
						CellVoltN_87_CAN:=FBRX_BMS_HCU_CELLV_22.oData[5]+SHL(BYTE_TO_INT(FBRX_BMS_HCU_CELLV_22.oData[4]),8);
						CellVoltN_88_CAN:=FBRX_BMS_HCU_CELLV_22.oData[7]+SHL(BYTE_TO_INT(FBRX_BMS_HCU_CELLV_22.oData[6]),8);
					
				ELSIF FBRX_BMS_HCU_CELLV_22 .oCanTimeout THEN										(* If timeout flag is enabled switch off LedRed *)
				 (*Crear los errores necesarios para cuando no se leen las variable despues del time out*)
						Counter_time_out_BATTERY:=Counter_time_out_BATTERY+1;
				END_IF
		FBRX_BMS_HCU_CELLV_23  (	iCAN			:= ADR(GVL.H_CAN_RX_6),  				(* Structure for sending / receiving CAN messages *)
								iCanId				:= 16#181650F3,							(* CAN Id of receiving message *) 
								iCanIdExtended		:= TRUE,  							(* Standard CAN Frame *)
								iTimeoutLimit		:= T#500MS,							(* Timeout after 500ms - Flag will be set *) 
								oByteCount			=> , 
								oData				=> , 
								oNewData			=> , 
								oCanTimeout			=> , 
								oReceiverId			=> , 
								oTooManyReceivers	=> );	
				
								
				IF FBRX_BMS_HCU_CELLV_23   .oNewData THEN											(* If new CAN data is available *)
						
						CellVoltN_89_CAN:=FBRX_BMS_HCU_CELLV_23.oData[1]+SHL(BYTE_TO_INT(FBRX_BMS_HCU_CELLV_23.oData[0]),8);
						CellVoltN_90_CAN:=FBRX_BMS_HCU_CELLV_23.oData[3]+SHL(BYTE_TO_INT(FBRX_BMS_HCU_CELLV_23.oData[2]),8);
						CellVoltN_91_CAN:=FBRX_BMS_HCU_CELLV_23.oData[5]+SHL(BYTE_TO_INT(FBRX_BMS_HCU_CELLV_23.oData[4]),8);
						CellVoltN_92_CAN:=FBRX_BMS_HCU_CELLV_23.oData[7]+SHL(BYTE_TO_INT(FBRX_BMS_HCU_CELLV_23.oData[6]),8);
					
				ELSIF FBRX_BMS_HCU_CELLV_23 .oCanTimeout THEN										(* If timeout flag is enabled switch off LedRed *)
				 (*Crear los errores necesarios para cuando no se leen las variable despues del time out*)
						Counter_time_out_BATTERY:=Counter_time_out_BATTERY+1;
				END_IF
		FBRX_BMS_HCU_CELLV_24  (	iCAN			:= ADR(GVL.H_CAN_RX_6),  				(* Structure for sending / receiving CAN messages *)
								iCanId				:= 16#181750F3,							(* CAN Id of receiving message *) 
								iCanIdExtended		:= TRUE,  							(* Standard CAN Frame *)
								iTimeoutLimit		:= T#500MS,							(* Timeout after 500ms - Flag will be set *) 
								oByteCount			=> , 
								oData				=> , 
								oNewData			=> , 
								oCanTimeout			=> , 
								oReceiverId			=> , 
								oTooManyReceivers	=> );	
				
								
				IF FBRX_BMS_HCU_CELLV_24   .oNewData THEN											(* If new CAN data is available *)
						
						CellVoltN_93_CAN:=FBRX_BMS_HCU_CELLV_24.oData[1]+SHL(BYTE_TO_INT(FBRX_BMS_HCU_CELLV_24.oData[0]),8);
						CellVoltN_94_CAN:=FBRX_BMS_HCU_CELLV_24.oData[3]+SHL(BYTE_TO_INT(FBRX_BMS_HCU_CELLV_24.oData[2]),8);
						CellVoltN_95_CAN:=FBRX_BMS_HCU_CELLV_24.oData[5]+SHL(BYTE_TO_INT(FBRX_BMS_HCU_CELLV_24.oData[4]),8);
						CellVoltN_96_CAN:=FBRX_BMS_HCU_CELLV_24.oData[7]+SHL(BYTE_TO_INT(FBRX_BMS_HCU_CELLV_24.oData[6]),8);
					
				ELSIF FBRX_BMS_HCU_CELLV_24 .oCanTimeout THEN										(* If timeout flag is enabled switch off LedRed *)
				 (*Crear los errores necesarios para cuando no se leen las variable despues del time out*)
						Counter_time_out_BATTERY:=Counter_time_out_BATTERY+1;
				END_IF
		FBRX_BMS_HCU_CELLV_25  (	iCAN			:= ADR(GVL.H_CAN_RX_6),  				(* Structure for sending / receiving CAN messages *)
								iCanId				:= 16#181850F3,							(* CAN Id of receiving message *) 
								iCanIdExtended		:= TRUE,  							(* Standard CAN Frame *)
								iTimeoutLimit		:= T#500MS,							(* Timeout after 500ms - Flag will be set *) 
								oByteCount			=> , 
								oData				=> , 
								oNewData			=> , 
								oCanTimeout			=> , 
								oReceiverId			=> , 
								oTooManyReceivers	=> );	
				
								
				IF FBRX_BMS_HCU_CELLV_25   .oNewData THEN											(* If new CAN data is available *)
						
						CellVoltN_97_CAN:=FBRX_BMS_HCU_CELLV_25.oData[1]+SHL(BYTE_TO_INT(FBRX_BMS_HCU_CELLV_25.oData[0]),8);
						CellVoltN_98_CAN:=FBRX_BMS_HCU_CELLV_25.oData[3]+SHL(BYTE_TO_INT(FBRX_BMS_HCU_CELLV_25.oData[2]),8);
						CellVoltN_99_CAN:=FBRX_BMS_HCU_CELLV_25.oData[5]+SHL(BYTE_TO_INT(FBRX_BMS_HCU_CELLV_25.oData[4]),8);
						CellVoltN_100_CAN:=FBRX_BMS_HCU_CELLV_25.oData[7]+SHL(BYTE_TO_INT(FBRX_BMS_HCU_CELLV_25.oData[6]),8);
					
				ELSIF FBRX_BMS_HCU_CELLV_25 .oCanTimeout THEN										(* If timeout flag is enabled switch off LedRed *)
				 (*Crear los errores necesarios para cuando no se leen las variable despues del time out*)
						Counter_time_out_BATTERY:=Counter_time_out_BATTERY+1;
				END_IF
		FBRX_BMS_HCU_CELLV_26  (	iCAN			:= ADR(GVL.H_CAN_RX_6),  				(* Structure for sending / receiving CAN messages *)
								iCanId				:= 16#181950F3,							(* CAN Id of receiving message *) 
								iCanIdExtended		:= TRUE,  							(* Standard CAN Frame *)
								iTimeoutLimit		:= T#500MS,							(* Timeout after 500ms - Flag will be set *) 
								oByteCount			=> , 
								oData				=> , 
								oNewData			=> , 
								oCanTimeout			=> , 
								oReceiverId			=> , 
								oTooManyReceivers	=> );	
				
								
				IF FBRX_BMS_HCU_CELLV_26   .oNewData THEN											(* If new CAN data is available *)
						
						CellVoltN_101_CAN:=FBRX_BMS_HCU_CELLV_26.oData[1]+SHL(BYTE_TO_INT(FBRX_BMS_HCU_CELLV_26.oData[0]),8);
						CellVoltN_102_CAN:=FBRX_BMS_HCU_CELLV_26.oData[3]+SHL(BYTE_TO_INT(FBRX_BMS_HCU_CELLV_26.oData[2]),8);
						CellVoltN_103_CAN:=FBRX_BMS_HCU_CELLV_26.oData[5]+SHL(BYTE_TO_INT(FBRX_BMS_HCU_CELLV_26.oData[4]),8);
						CellVoltN_104_CAN:=FBRX_BMS_HCU_CELLV_26.oData[7]+SHL(BYTE_TO_INT(FBRX_BMS_HCU_CELLV_26.oData[6]),8);
					
				ELSIF FBRX_BMS_HCU_CELLV_26 .oCanTimeout THEN										(* If timeout flag is enabled switch off LedRed *)
				 (*Crear los errores necesarios para cuando no se leen las variable despues del time out*)
						Counter_time_out_BATTERY:=Counter_time_out_BATTERY+1;
				END_IF
				
		FBRX_BMS_HCU_CELLV_27  (	iCAN			:= ADR(GVL.H_CAN_RX_6),  				(* Structure for sending / receiving CAN messages *)
								iCanId				:= 16#181A50F3,							(* CAN Id of receiving message *) 
								iCanIdExtended		:= TRUE,  							(* Standard CAN Frame *)
								iTimeoutLimit		:= T#500MS,							(* Timeout after 500ms - Flag will be set *) 
								oByteCount			=> , 
								oData				=> , 
								oNewData			=> , 
								oCanTimeout			=> , 
								oReceiverId			=> , 
								oTooManyReceivers	=> );	
				
								
				IF FBRX_BMS_HCU_CELLV_27   .oNewData THEN											(* If new CAN data is available *)
						
						CellVoltN_105_CAN:=FBRX_BMS_HCU_CELLV_27.oData[1]+SHL(BYTE_TO_INT(FBRX_BMS_HCU_CELLV_27.oData[0]),8);
						CellVoltN_106_CAN:=FBRX_BMS_HCU_CELLV_27.oData[3]+SHL(BYTE_TO_INT(FBRX_BMS_HCU_CELLV_27.oData[2]),8);
						CellVoltN_107_CAN:=FBRX_BMS_HCU_CELLV_27.oData[5]+SHL(BYTE_TO_INT(FBRX_BMS_HCU_CELLV_27.oData[4]),8);
						CellVoltN_108_CAN:=FBRX_BMS_HCU_CELLV_27.oData[7]+SHL(BYTE_TO_INT(FBRX_BMS_HCU_CELLV_27.oData[6]),8);
					
				ELSIF FBRX_BMS_HCU_CELLV_27 .oCanTimeout THEN										(* If timeout flag is enabled switch off LedRed *)
				 (*Crear los errores necesarios para cuando no se leen las variable despues del time out*)
						Counter_time_out_BATTERY:=Counter_time_out_BATTERY+1;
				END_IF
				
		FBRX_BMS_HCU_CELLV_28  (	iCAN			:= ADR(GVL.H_CAN_RX_6),  				(* Structure for sending / receiving CAN messages *)
								iCanId				:= 16#181B50F3,							(* CAN Id of receiving message *) 
								iCanIdExtended		:= TRUE,  							(* Standard CAN Frame *)
								iTimeoutLimit		:= T#500MS,							(* Timeout after 500ms - Flag will be set *) 
								oByteCount			=> , 
								oData				=> , 
								oNewData			=> , 
								oCanTimeout			=> , 
								oReceiverId			=> , 
								oTooManyReceivers	=> );	
				
								
				IF FBRX_BMS_HCU_CELLV_28   .oNewData THEN											(* If new CAN data is available *)
						
						CellVoltN_109_CAN:=FBRX_BMS_HCU_CELLV_28.oData[1]+SHL(BYTE_TO_INT(FBRX_BMS_HCU_CELLV_28.oData[0]),8);
						CellVoltN_110_CAN:=FBRX_BMS_HCU_CELLV_28.oData[3]+SHL(BYTE_TO_INT(FBRX_BMS_HCU_CELLV_28.oData[2]),8);
						CellVoltN_111_CAN:=FBRX_BMS_HCU_CELLV_28.oData[5]+SHL(BYTE_TO_INT(FBRX_BMS_HCU_CELLV_28.oData[4]),8);
						CellVoltN_112_CAN:=FBRX_BMS_HCU_CELLV_28.oData[7]+SHL(BYTE_TO_INT(FBRX_BMS_HCU_CELLV_28.oData[6]),8);
					
				ELSIF FBRX_BMS_HCU_CELLV_28 .oCanTimeout THEN										(* If timeout flag is enabled switch off LedRed *)
				 (*Crear los errores necesarios para cuando no se leen las variable despues del time out*)
						Counter_time_out_BATTERY:=Counter_time_out_BATTERY+1;
				END_IF
				
				
		FBRX_BMS_HCU_CELLV_29  (	iCAN			:= ADR(GVL.H_CAN_RX_6),  				(* Structure for sending / receiving CAN messages *)
								iCanId				:= 16#181C50F3,							(* CAN Id of receiving message *) 
								iCanIdExtended		:= TRUE,  							(* Standard CAN Frame *)
								iTimeoutLimit		:= T#500MS,							(* Timeout after 500ms - Flag will be set *) 
								oByteCount			=> , 
								oData				=> , 
								oNewData			=> , 
								oCanTimeout			=> , 
								oReceiverId			=> , 
								oTooManyReceivers	=> );	
				
								
				IF FBRX_BMS_HCU_CELLV_29   .oNewData THEN											(* If new CAN data is available *)
						
						CellVoltN_113_CAN:=FBRX_BMS_HCU_CELLV_29.oData[1]+SHL(BYTE_TO_INT(FBRX_BMS_HCU_CELLV_29.oData[0]),8);
						CellVoltN_114_CAN:=FBRX_BMS_HCU_CELLV_29.oData[3]+SHL(BYTE_TO_INT(FBRX_BMS_HCU_CELLV_29.oData[2]),8);
						CellVoltN_115_CAN:=FBRX_BMS_HCU_CELLV_29.oData[5]+SHL(BYTE_TO_INT(FBRX_BMS_HCU_CELLV_29.oData[4]),8);
						CellVoltN_116_CAN:=FBRX_BMS_HCU_CELLV_29.oData[7]+SHL(BYTE_TO_INT(FBRX_BMS_HCU_CELLV_29.oData[6]),8);
					
				ELSIF FBRX_BMS_HCU_CELLV_29 .oCanTimeout THEN										(* If timeout flag is enabled switch off LedRed *)
				 (*Crear los errores necesarios para cuando no se leen las variable despues del time out*)
						Counter_time_out_BATTERY:=Counter_time_out_BATTERY+1;
				END_IF
				
				
		FBRX_BMS_HCU_CELLV_30  (	iCAN			:= ADR(GVL.H_CAN_RX_6),  				(* Structure for sending / receiving CAN messages *)
								iCanId				:= 16#181D50F3,							(* CAN Id of receiving message *) 
								iCanIdExtended		:= TRUE,  							(* Standard CAN Frame *)
								iTimeoutLimit		:= T#500MS,							(* Timeout after 500ms - Flag will be set *) 
								oByteCount			=> , 
								oData				=> , 
								oNewData			=> , 
								oCanTimeout			=> , 
								oReceiverId			=> , 
								oTooManyReceivers	=> );	
				
								
				IF FBRX_BMS_HCU_CELLV_30   .oNewData THEN											(* If new CAN data is available *)
						
						CellVoltN_117_CAN:=FBRX_BMS_HCU_CELLV_30.oData[1]+SHL(BYTE_TO_INT(FBRX_BMS_HCU_CELLV_30.oData[0]),8);
						CellVoltN_118_CAN:=FBRX_BMS_HCU_CELLV_30.oData[3]+SHL(BYTE_TO_INT(FBRX_BMS_HCU_CELLV_30.oData[2]),8);
						CellVoltN_119_CAN:=FBRX_BMS_HCU_CELLV_30.oData[5]+SHL(BYTE_TO_INT(FBRX_BMS_HCU_CELLV_30.oData[4]),8);
						CellVoltN_120_CAN:=FBRX_BMS_HCU_CELLV_30.oData[7]+SHL(BYTE_TO_INT(FBRX_BMS_HCU_CELLV_30.oData[6]),8);
					
				ELSIF FBRX_BMS_HCU_CELLV_30 .oCanTimeout THEN										(* If timeout flag is enabled switch off LedRed *)
				 (*Crear los errores necesarios para cuando no se leen las variable despues del time out*)
						Counter_time_out_BATTERY:=Counter_time_out_BATTERY+1;
				END_IF
				
				
		FBRX_BMS_HCU_CELLV_31  (	iCAN			:= ADR(GVL.H_CAN_RX_6),  				(* Structure for sending / receiving CAN messages *)
								iCanId				:= 16#181E50F3,							(* CAN Id of receiving message *) 
								iCanIdExtended		:= TRUE,  							(* Standard CAN Frame *)
								iTimeoutLimit		:= T#500MS,							(* Timeout after 500ms - Flag will be set *) 
								oByteCount			=> , 
								oData				=> , 
								oNewData			=> , 
								oCanTimeout			=> , 
								oReceiverId			=> , 
								oTooManyReceivers	=> );	
				
								
				IF FBRX_BMS_HCU_CELLV_31   .oNewData THEN											(* If new CAN data is available *)
						
						CellVoltN_121_CAN:=FBRX_BMS_HCU_CELLV_31.oData[1]+SHL(BYTE_TO_INT(FBRX_BMS_HCU_CELLV_31.oData[0]),8);
						CellVoltN_122_CAN:=FBRX_BMS_HCU_CELLV_31.oData[3]+SHL(BYTE_TO_INT(FBRX_BMS_HCU_CELLV_31.oData[2]),8);
						CellVoltN_123_CAN:=FBRX_BMS_HCU_CELLV_31.oData[5]+SHL(BYTE_TO_INT(FBRX_BMS_HCU_CELLV_31.oData[4]),8);
						CellVoltN_124_CAN:=FBRX_BMS_HCU_CELLV_31.oData[7]+SHL(BYTE_TO_INT(FBRX_BMS_HCU_CELLV_31.oData[6]),8);
					
				ELSIF FBRX_BMS_HCU_CELLV_31 .oCanTimeout THEN										(* If timeout flag is enabled switch off LedRed *)
				 (*Crear los errores necesarios para cuando no se leen las variable despues del time out*)
						Counter_time_out_BATTERY:=Counter_time_out_BATTERY+1;
				END_IF
				
		FBRX_BMS_HCU_CELLV_32  (	iCAN			:= ADR(GVL.H_CAN_RX_6),  				(* Structure for sending / receiving CAN messages *)
								iCanId				:= 16#181F50F3,							(* CAN Id of receiving message *) 
								iCanIdExtended		:= TRUE,  							(* Standard CAN Frame *)
								iTimeoutLimit		:= T#500MS,							(* Timeout after 500ms - Flag will be set *) 
								oByteCount			=> , 
								oData				=> , 
								oNewData			=> , 
								oCanTimeout			=> , 
								oReceiverId			=> , 
								oTooManyReceivers	=> );	
				
								
				IF FBRX_BMS_HCU_CELLV_32   .oNewData THEN											(* If new CAN data is available *)
						
						CellVoltN_125_CAN:=FBRX_BMS_HCU_CELLV_32.oData[1]+SHL(BYTE_TO_INT(FBRX_BMS_HCU_CELLV_32.oData[0]),8);
						CellVoltN_126_CAN:=FBRX_BMS_HCU_CELLV_32.oData[3]+SHL(BYTE_TO_INT(FBRX_BMS_HCU_CELLV_32.oData[2]),8);
						CellVoltN_127_CAN:=FBRX_BMS_HCU_CELLV_32.oData[5]+SHL(BYTE_TO_INT(FBRX_BMS_HCU_CELLV_32.oData[4]),8);
						CellVoltN_128_CAN:=FBRX_BMS_HCU_CELLV_32.oData[7]+SHL(BYTE_TO_INT(FBRX_BMS_HCU_CELLV_32.oData[6]),8);
					
				ELSIF FBRX_BMS_HCU_CELLV_32 .oCanTimeout THEN										(* If timeout flag is enabled switch off LedRed *)
				 (*Crear los errores necesarios para cuando no se leen las variable despues del time out*)
						Counter_time_out_BATTERY:=Counter_time_out_BATTERY+1;
				END_IF
				
				
		FBRX_BMS_HCU_CELLV_33  (	iCAN			:= ADR(GVL.H_CAN_RX_6),  				(* Structure for sending / receiving CAN messages *)
								iCanId				:= 16#182050F3,							(* CAN Id of receiving message *) 
								iCanIdExtended		:= TRUE,  							(* Standard CAN Frame *)
								iTimeoutLimit		:= T#500MS,							(* Timeout after 500ms - Flag will be set *) 
								oByteCount			=> , 
								oData				=> , 
								oNewData			=> , 
								oCanTimeout			=> , 
								oReceiverId			=> , 
								oTooManyReceivers	=> );	
				
								
				IF FBRX_BMS_HCU_CELLV_33   .oNewData THEN											(* If new CAN data is available *)
						
						CellVoltN_129_CAN:=FBRX_BMS_HCU_CELLV_33.oData[1]+SHL(BYTE_TO_INT(FBRX_BMS_HCU_CELLV_33.oData[0]),8);
						CellVoltN_130_CAN:=FBRX_BMS_HCU_CELLV_33.oData[3]+SHL(BYTE_TO_INT(FBRX_BMS_HCU_CELLV_33.oData[2]),8);
						CellVoltN_131_CAN:=FBRX_BMS_HCU_CELLV_33.oData[5]+SHL(BYTE_TO_INT(FBRX_BMS_HCU_CELLV_33.oData[4]),8);
						CellVoltN_132_CAN:=FBRX_BMS_HCU_CELLV_33.oData[7]+SHL(BYTE_TO_INT(FBRX_BMS_HCU_CELLV_33.oData[6]),8);
					
				ELSIF FBRX_BMS_HCU_CELLV_33 .oCanTimeout THEN										(* If timeout flag is enabled switch off LedRed *)
				 (*Crear los errores necesarios para cuando no se leen las variable despues del time out*)
						Counter_time_out_BATTERY:=Counter_time_out_BATTERY+1;
				END_IF
				
				
		FBRX_BMS_HCU_CELLV_34  (	iCAN			:= ADR(GVL.H_CAN_RX_6),  				(* Structure for sending / receiving CAN messages *)
								iCanId				:= 16#182150F3,							(* CAN Id of receiving message *) 
								iCanIdExtended		:= TRUE,  							(* Standard CAN Frame *)
								iTimeoutLimit		:= T#500MS,							(* Timeout after 500ms - Flag will be set *) 
								oByteCount			=> , 
								oData				=> , 
								oNewData			=> , 
								oCanTimeout			=> , 
								oReceiverId			=> , 
								oTooManyReceivers	=> );	
				
								
				IF FBRX_BMS_HCU_CELLV_34   .oNewData THEN											(* If new CAN data is available *)
						
						CellVoltN_133_CAN:=FBRX_BMS_HCU_CELLV_34.oData[1]+SHL(BYTE_TO_INT(FBRX_BMS_HCU_CELLV_34.oData[0]),8);
						CellVoltN_134_CAN:=FBRX_BMS_HCU_CELLV_34.oData[3]+SHL(BYTE_TO_INT(FBRX_BMS_HCU_CELLV_34.oData[2]),8);
						CellVoltN_135_CAN:=FBRX_BMS_HCU_CELLV_34.oData[5]+SHL(BYTE_TO_INT(FBRX_BMS_HCU_CELLV_34.oData[4]),8);
						CellVoltN_136_CAN:=FBRX_BMS_HCU_CELLV_34.oData[7]+SHL(BYTE_TO_INT(FBRX_BMS_HCU_CELLV_34.oData[6]),8);
					
				ELSIF FBRX_BMS_HCU_CELLV_34 .oCanTimeout THEN										(* If timeout flag is enabled switch off LedRed *)
				 (*Crear los errores necesarios para cuando no se leen las variable despues del time out*)
						Counter_time_out_BATTERY:=Counter_time_out_BATTERY+1;
				END_IF
				
				
		FBRX_BMS_HCU_CELLV_35  (	iCAN			:= ADR(GVL.H_CAN_RX_6),  				(* Structure for sending / receiving CAN messages *)
								iCanId				:= 16#182250F3,							(* CAN Id of receiving message *) 
								iCanIdExtended		:= TRUE,  							(* Standard CAN Frame *)
								iTimeoutLimit		:= T#500MS,							(* Timeout after 500ms - Flag will be set *) 
								oByteCount			=> , 
								oData				=> , 
								oNewData			=> , 
								oCanTimeout			=> , 
								oReceiverId			=> , 
								oTooManyReceivers	=> );	
				
								
				IF FBRX_BMS_HCU_CELLV_35   .oNewData THEN											(* If new CAN data is available *)
						
						CellVoltN_137_CAN:=FBRX_BMS_HCU_CELLV_35.oData[1]+SHL(BYTE_TO_INT(FBRX_BMS_HCU_CELLV_35.oData[0]),8);
						CellVoltN_138_CAN:=FBRX_BMS_HCU_CELLV_35.oData[3]+SHL(BYTE_TO_INT(FBRX_BMS_HCU_CELLV_35.oData[2]),8);
						
				ELSIF FBRX_BMS_HCU_CELLV_35 .oCanTimeout THEN										(* If timeout flag is enabled switch off LedRed *)
				 (*Crear los errores necesarios para cuando no se leen las variable despues del time out*)
						Counter_time_out_BATTERY:=Counter_time_out_BATTERY+1;
				END_IF
				
				
		FBRX_BMS_HCU_CELLT_1  (	iCAN			:= ADR(GVL.H_CAN_RX_6),  				(* Structure for sending / receiving CAN messages *)
								iCanId				:= 16#185050F3,							(* CAN Id of receiving message *) 
								iCanIdExtended		:= TRUE,  							(* Standard CAN Frame *)
								iTimeoutLimit		:= T#500MS,							(* Timeout after 500ms - Flag will be set *) 
								oByteCount			=> , 
								oData				=> , 
								oNewData			=> , 
								oCanTimeout			=> , 
								oReceiverId			=> , 
								oTooManyReceivers	=> );	
				
								
				IF FBRX_BMS_HCU_CELLT_1   .oNewData THEN											(* If new CAN data is available *)
						
						CellTempN_1_CAN:=FBRX_BMS_HCU_CELLT_1.oData[0];
						CellTempN_2_CAN:=FBRX_BMS_HCU_CELLT_1.oData[1];
						CellTempN_3_CAN:=FBRX_BMS_HCU_CELLT_1.oData[2];
						CellTempN_4_CAN:=FBRX_BMS_HCU_CELLT_1.oData[3];
						CellTempN_5_CAN:=FBRX_BMS_HCU_CELLT_1.oData[4];
						CellTempN_6_CAN:=FBRX_BMS_HCU_CELLT_1.oData[5];
						CellTempN_7_CAN:=FBRX_BMS_HCU_CELLT_1.oData[6];
						CellTempN_8_CAN:=FBRX_BMS_HCU_CELLT_1.oData[7];
						
				ELSIF FBRX_BMS_HCU_CELLT_1 .oCanTimeout THEN										(* If timeout flag is enabled switch off LedRed *)
				 (*Crear los errores necesarios para cuando no se leen las variable despues del time out*)
						Counter_time_out_BATTERY:=Counter_time_out_BATTERY+1;
				END_IF
				
				
		FBRX_BMS_HCU_CELLT_2  (	iCAN			:= ADR(GVL.H_CAN_RX_6),  				(* Structure for sending / receiving CAN messages *)
								iCanId				:= 16#185250F3,							(* CAN Id of receiving message *) 
								iCanIdExtended		:= TRUE,  							(* Standard CAN Frame *)
								iTimeoutLimit		:= T#500MS,							(* Timeout after 500ms - Flag will be set *) 
								oByteCount			=> , 
								oData				=> , 
								oNewData			=> , 
								oCanTimeout			=> , 
								oReceiverId			=> , 
								oTooManyReceivers	=> );	
				
								
				IF FBRX_BMS_HCU_CELLT_2   .oNewData THEN											(* If new CAN data is available *)
						
						CellTempN_9_CAN:=FBRX_BMS_HCU_CELLT_2.oData[0];
						CellTempN_10_CAN:=FBRX_BMS_HCU_CELLT_2.oData[1];
						CellTempN_11_CAN:=FBRX_BMS_HCU_CELLT_2.oData[2];
						CellTempN_12_CAN:=FBRX_BMS_HCU_CELLT_2.oData[3];
						CellTempN_13_CAN:=FBRX_BMS_HCU_CELLT_2.oData[4];
						CellTempN_14_CAN:=FBRX_BMS_HCU_CELLT_2.oData[5];
						CellTempN_15_CAN:=FBRX_BMS_HCU_CELLT_2.oData[6];
						CellTempN_16_CAN:=FBRX_BMS_HCU_CELLT_2.oData[7];
						
				ELSIF FBRX_BMS_HCU_CELLT_2 .oCanTimeout THEN										(* If timeout flag is enabled switch off LedRed *)
				 (*Crear los errores necesarios para cuando no se leen las variable despues del time out*)
						Counter_time_out_BATTERY:=Counter_time_out_BATTERY+1;
				END_IF
				
				
		FBRX_BMS_HCU_CELLT_3  (	iCAN			:= ADR(GVL.H_CAN_RX_6),  				(* Structure for sending / receiving CAN messages *)
								iCanId				:= 16#185450F3,							(* CAN Id of receiving message *) 
								iCanIdExtended		:= TRUE,  							(* Standard CAN Frame *)
								iTimeoutLimit		:= T#500MS,							(* Timeout after 500ms - Flag will be set *) 
								oByteCount			=> , 
								oData				=> , 
								oNewData			=> , 
								oCanTimeout			=> , 
								oReceiverId			=> , 
								oTooManyReceivers	=> );	
				
								
				IF FBRX_BMS_HCU_CELLT_3   .oNewData THEN											(* If new CAN data is available *)
						
						CellTempN_17_CAN:=FBRX_BMS_HCU_CELLT_3.oData[0];
						CellTempN_18_CAN:=FBRX_BMS_HCU_CELLT_3.oData[1];
						CellTempN_19_CAN:=FBRX_BMS_HCU_CELLT_3.oData[2];
						CellTempN_20_CAN:=FBRX_BMS_HCU_CELLT_3.oData[3];
						CellTempN_21_CAN:=FBRX_BMS_HCU_CELLT_3.oData[4];
						CellTempN_22_CAN:=FBRX_BMS_HCU_CELLT_3.oData[5];
						CellTempN_23_CAN:=FBRX_BMS_HCU_CELLT_3.oData[6];
						CellTempN_24_CAN:=FBRX_BMS_HCU_CELLT_3.oData[7];
						
				ELSIF FBRX_BMS_HCU_CELLT_3 .oCanTimeout THEN										(* If timeout flag is enabled switch off LedRed *)
				 (*Crear los errores necesarios para cuando no se leen las variable despues del time out*)
						Counter_time_out_BATTERY:=Counter_time_out_BATTERY+1;
				END_IF
				
				
		FBRX_BMS_HCU_CELLT_4  (	iCAN			:= ADR(GVL.H_CAN_RX_6),  				(* Structure for sending / receiving CAN messages *)
								iCanId				:= 16#185650F3,							(* CAN Id of receiving message *) 
								iCanIdExtended		:= TRUE,  							(* Standard CAN Frame *)
								iTimeoutLimit		:= T#500MS,							(* Timeout after 500ms - Flag will be set *) 
								oByteCount			=> , 
								oData				=> , 
								oNewData			=> , 
								oCanTimeout			=> , 
								oReceiverId			=> , 
								oTooManyReceivers	=> );	
				
								
				IF FBRX_BMS_HCU_CELLT_4   .oNewData THEN											(* If new CAN data is available *)
						
						CellTempN_25_CAN:=FBRX_BMS_HCU_CELLT_4.oData[0];
						CellTempN_26_CAN:=FBRX_BMS_HCU_CELLT_4.oData[1];
						CellTempN_27_CAN:=FBRX_BMS_HCU_CELLT_4.oData[2];
						CellTempN_28_CAN:=FBRX_BMS_HCU_CELLT_4.oData[3];
						CellTempN_29_CAN:=FBRX_BMS_HCU_CELLT_4.oData[4];
						CellTempN_30_CAN:=FBRX_BMS_HCU_CELLT_4.oData[5];
						CellTempN_31_CAN:=FBRX_BMS_HCU_CELLT_4.oData[6];
						CellTempN_32_CAN:=FBRX_BMS_HCU_CELLT_4.oData[7];
						
				ELSIF FBRX_BMS_HCU_CELLT_4 .oCanTimeout THEN										(* If timeout flag is enabled switch off LedRed *)
				 (*Crear los errores necesarios para cuando no se leen las variable despues del time out*)
						Counter_time_out_BATTERY:=Counter_time_out_BATTERY+1;
				END_IF
				
				
		FBRX_BMS_HCU_CELLT_5  (	iCAN			:= ADR(GVL.H_CAN_RX_6),  				(* Structure for sending / receiving CAN messages *)
								iCanId				:= 16#185850F3,							(* CAN Id of receiving message *) 
								iCanIdExtended		:= TRUE,  							(* Standard CAN Frame *)
								iTimeoutLimit		:= T#500MS,							(* Timeout after 500ms - Flag will be set *) 
								oByteCount			=> , 
								oData				=> , 
								oNewData			=> , 
								oCanTimeout			=> , 
								oReceiverId			=> , 
								oTooManyReceivers	=> );	
				
								
				IF FBRX_BMS_HCU_CELLT_5   .oNewData THEN											(* If new CAN data is available *)
						
						CellTempN_33_CAN:=FBRX_BMS_HCU_CELLT_5.oData[0];
						CellTempN_34_CAN:=FBRX_BMS_HCU_CELLT_5.oData[1];
						CellTempN_35_CAN:=FBRX_BMS_HCU_CELLT_5.oData[2];
						CellTempN_36_CAN:=FBRX_BMS_HCU_CELLT_5.oData[3];
						CellTempN_37_CAN:=FBRX_BMS_HCU_CELLT_5.oData[4];
						CellTempN_38_CAN:=FBRX_BMS_HCU_CELLT_5.oData[5];
						CellTempN_39_CAN:=FBRX_BMS_HCU_CELLT_5.oData[6];
						CellTempN_40_CAN:=FBRX_BMS_HCU_CELLT_5.oData[7];
						
				ELSIF FBRX_BMS_HCU_CELLT_5 .oCanTimeout THEN										(* If timeout flag is enabled switch off LedRed *)
				 (*Crear los errores necesarios para cuando no se leen las variable despues del time out*)
						Counter_time_out_BATTERY:=Counter_time_out_BATTERY+1;
				END_IF
				
				
		FBRX_BMS_HCU_CELLT_6  (	iCAN			:= ADR(GVL.H_CAN_RX_6),  				(* Structure for sending / receiving CAN messages *)
								iCanId				:= 16#185A50F3,							(* CAN Id of receiving message *) 
								iCanIdExtended		:= TRUE,  							(* Standard CAN Frame *)
								iTimeoutLimit		:= T#500MS,							(* Timeout after 500ms - Flag will be set *) 
								oByteCount			=> , 
								oData				=> , 
								oNewData			=> , 
								oCanTimeout			=> , 
								oReceiverId			=> , 
								oTooManyReceivers	=> );	
				
								
				IF FBRX_BMS_HCU_CELLT_6   .oNewData THEN											(* If new CAN data is available *)
						
						CellTempN_41_CAN:=FBRX_BMS_HCU_CELLT_6.oData[0];
						CellTempN_42_CAN:=FBRX_BMS_HCU_CELLT_6.oData[1];
						CellTempN_43_CAN:=FBRX_BMS_HCU_CELLT_6.oData[2];
						CellTempN_44_CAN:=FBRX_BMS_HCU_CELLT_6.oData[3];
						CellTempN_45_CAN:=FBRX_BMS_HCU_CELLT_6.oData[4];
						CellTempN_46_CAN:=FBRX_BMS_HCU_CELLT_6.oData[5];
						CellTempN_47_CAN:=FBRX_BMS_HCU_CELLT_6.oData[6];
						CellTempN_48_CAN:=FBRX_BMS_HCU_CELLT_6.oData[7];
						
				ELSIF FBRX_BMS_HCU_CELLT_6 .oCanTimeout THEN										(* If timeout flag is enabled switch off LedRed *)
				 (*Crear los errores necesarios para cuando no se leen las variable despues del time out*)
						Counter_time_out_BATTERY:=Counter_time_out_BATTERY+1;
				END_IF
				
				
		FBRX_BMS_HCU_CELLT_7  (	iCAN			:= ADR(GVL.H_CAN_RX_6),  				(* Structure for sending / receiving CAN messages *)
								iCanId				:= 16#185C50F3,							(* CAN Id of receiving message *) 
								iCanIdExtended		:= TRUE,  							(* Standard CAN Frame *)
								iTimeoutLimit		:= T#500MS,							(* Timeout after 500ms - Flag will be set *) 
								oByteCount			=> , 
								oData				=> , 
								oNewData			=> , 
								oCanTimeout			=> , 
								oReceiverId			=> , 
								oTooManyReceivers	=> );	
				
								
				IF FBRX_BMS_HCU_CELLT_7   .oNewData THEN											(* If new CAN data is available *)
						
						CellTempN_49_CAN:=FBRX_BMS_HCU_CELLT_7.oData[0];
						CellTempN_50_CAN:=FBRX_BMS_HCU_CELLT_7.oData[1];
						CellTempN_51_CAN:=FBRX_BMS_HCU_CELLT_7.oData[2];
						CellTempN_52_CAN:=FBRX_BMS_HCU_CELLT_7.oData[3];
						CellTempN_53_CAN:=FBRX_BMS_HCU_CELLT_7.oData[4];
						CellTempN_54_CAN:=FBRX_BMS_HCU_CELLT_7.oData[5];
						CellTempN_55_CAN:=FBRX_BMS_HCU_CELLT_7.oData[6];
						CellTempN_56_CAN:=FBRX_BMS_HCU_CELLT_7.oData[7];
						
				ELSIF FBRX_BMS_HCU_CELLT_7 .oCanTimeout THEN										(* If timeout flag is enabled switch off LedRed *)
				 (*Crear los errores necesarios para cuando no se leen las variable despues del time out*)
						Counter_time_out_BATTERY:=Counter_time_out_BATTERY+1;
				END_IF
				
				
		FBRX_BMS_HCU_CELLT_8  (	iCAN			:= ADR(GVL.H_CAN_RX_6),  				(* Structure for sending / receiving CAN messages *)
								iCanId				:= 16#185E50F3,							(* CAN Id of receiving message *) 
								iCanIdExtended		:= TRUE,  							(* Standard CAN Frame *)
								iTimeoutLimit		:= T#500MS,							(* Timeout after 500ms - Flag will be set *) 
								oByteCount			=> , 
								oData				=> , 
								oNewData			=> , 
								oCanTimeout			=> , 
								oReceiverId			=> , 
								oTooManyReceivers	=> );	
				
								
				IF FBRX_BMS_HCU_CELLT_8   .oNewData THEN											(* If new CAN data is available *)
						
						CellTempN_57_CAN:=FBRX_BMS_HCU_CELLT_8.oData[0];
						CellTempN_58_CAN:=FBRX_BMS_HCU_CELLT_8.oData[1];
						CellTempN_59_CAN:=FBRX_BMS_HCU_CELLT_8.oData[2];
						CellTempN_60_CAN:=FBRX_BMS_HCU_CELLT_8.oData[3];
						
						
				ELSIF FBRX_BMS_HCU_CELLT_8 .oCanTimeout THEN										(* If timeout flag is enabled switch off LedRed *)
				 (*Crear los errores necesarios para cuando no se leen las variable despues del time out*)
						Counter_time_out_BATTERY:=Counter_time_out_BATTERY+1;
				END_IF
				
				
		FBRX_BMS_HCU_CMD  (	iCAN			:= ADR(GVL.H_CAN_RX_6),  				(* Structure for sending / receiving CAN messages *)
								iCanId				:= 16#1801F340,							(* CAN Id of receiving message *) 
								iCanIdExtended		:= TRUE,  							(* Standard CAN Frame *)
								iTimeoutLimit		:= T#500MS,							(* Timeout after 500ms - Flag will be set *) 
								oByteCount			=> , 
								oData				=> , 
								oNewData			=> , 
								oCanTimeout			=> , 
								oReceiverId			=> , 
								oTooManyReceivers	=> );	
				
								
				IF FBRX_BMS_HCU_CMD   .oNewData THEN											(* If new CAN data is available *)
						
						MainRlyCmd_CAN:=FBRX_BMS_HCU_CMD.oData[0];
						ShutDownCmd_CAN:=FBRX_BMS_HCU_CMD.oData[1];
												
						
				ELSIF FBRX_BMS_HCU_CMD .oCanTimeout THEN										(* If timeout flag is enabled switch off LedRed *)
				 (*Crear los errores necesarios para cuando no se leen las variable despues del time out*)
						Counter_time_out_BATTERY:=Counter_time_out_BATTERY+1;
				END_IF
				
(*-----------------------------------------------FIN_BATTERY_RX--------------------------------------------------*)

*)

END_FUNCTION_BLOCK

// Device/Application/UPM03/CAN_TX_V_1_4

(* 2019/06/25	VERSION V1_1 : Introduccion de la linea de CAN de la AIM para enviar datos de estados de la EVCU *)

FUNCTION_BLOCK CAN_TX_V_1_4
VAR_INPUT
	
	
		Brake_Light_CAN: BOOL;
		Pre_Charge_CAN: BOOL;
		Estado_CAN: LREAL;
		Info_Inverter_Error_CAN: UINT;
		Estado_Error_CAN: LREAL;
		Throttle_CAN: REAL;
				
		AIM_TempMotor1_CAN: USINT;
		AIM_TempInverter1_CAN: USINT; 
		AIM_TempMotor2_CAN: USINT;
		AIM_TempInverter2_CAN: USINT;
		AIM_TempMotor3_CAN: USINT;
		AIM_TempInverter3_CAN: USINT;
		AIM_TempMotor4_CAN: USINT;
		AIM_TempInverter4_CAN: USINT;
		
		AIM_bError1_CAN: BOOL;
		AIM_bError2_CAN: BOOL;
		AIM_bError3_CAN: BOOL;
		AIM_bError4_CAN: BOOL;
		
				
		AIM_TempIGBT1_CAN: USINT;
		AIM_TempIGBT2_CAN: USINT;
		AIM_TempIGBT3_CAN: USINT;
		AIM_TempIGBT4_CAN: USINT;
		
		AIM_bDerating1_CAN: BOOL;
		AIM_bDerating2_CAN: BOOL;
		AIM_bDerating3_CAN: BOOL;
		AIM_bDerating4_CAN: BOOL;
		
		K15_Value: WORD;
		
		AIM_TorqueCurrent1_CAN: INT;
		AIM_TorqueCurrent2_CAN: INT;
		AIM_TorqueCurrent3_CAN: INT;
		AIM_TorqueCurrent4_CAN: INT;
		
		AIM_MagnetizingCurrent1_CAN: INT;
		AIM_MagnetizingCurrent2_CAN: INT;
		AIM_MagnetizingCurrent3_CAN: INT;
		AIM_MagnetizingCurrent4_CAN: INT;
		
		AIM_TargetVelocity1_CAN: INT;
		AIM_TargetVelocity2_CAN: INT;
		AIM_TargetVelocity3_CAN: INT;
		AIM_TargetVelocity4_CAN: INT;
			
		AIM_TorqueLimitPositiv1_CAN: INT;
		AIM_TorqueLimitPositiv2_CAN: INT;
		AIM_TorqueLimitPositiv3_CAN: INT;
		AIM_TorqueLimitPositiv4_CAN: INT;
		
		AIM_ActualVelocity1_CAN: INT;
		AIM_ActualVelocity2_CAN: INT;
		AIM_ActualVelocity3_CAN: INT;
		AIM_ActualVelocity4_CAN: INT;
				
		
		AIM_YC_TorqueLimitPositiv1_CAN: INT;
		AIM_YC_TorqueLimitPositiv2_CAN: INT;
		AIM_YC_TorqueLimitPositiv3_CAN: INT;
		AIM_YC_TorqueLimitPositiv4_CAN: INT;
				
		Speed_RPM_CAN: REAL;
		
		AIM_ErrorInfo1_CAN: UINT;
		AIM_ErrorInfo2_CAN: UINT;
		AIM_ErrorInfo3_CAN: UINT;
		AIM_ErrorInfo4_CAN: UINT;
		
END_VAR
VAR_OUTPUT
END_VAR
VAR
(*CanTX*) 

	(*Auxiliary Variable*)
		TxData: ARRAY [0..7]OF BYTE;
	
	(*AIM*)	
		FBTX_AIM_1:CanTx;              (* Function block to send one CAN message *)
		
		FBTX_AIM_2:CanTx;	
	
		FBTX_AIM_3:CanTx;

		FBTX_AIM_4:CanTx;

		FBTX_AIM_5:CanTx;

		FBTX_AIM_6:CanTx;

		FBTX_AIM_7:CanTx;

		FBTX_AIM_8:CanTx;	

		FBTX_AIM_9:CanTx;

		FBTX_AIM_10:CanTx;

		FBTX_AIM_11:CanTx;	

END_VAR

